C05479=1233.629,-83.711,-36.665,179.745,5.254,148.987
C05480=1233.634,-83.960,-36.654,179.743,5.255,148.988
C05481=1233.639,-84.210,-36.643,179.740,5.254,148.989
C05482=1233.645,-84.460,-36.632,179.738,5.255,148.989
C05483=1233.649,-84.710,-36.620,179.735,5.254,148.990
C05484=1233.655,-84.959,-36.609,179.733,5.254,148.991
C05485=1233.660,-85.209,-36.597,179.730,5.254,148.991
C05486=1233.665,-85.459,-36.587,179.728,5.254,148.992
C05487=1233.670,-85.709,-36.576,179.726,5.254,148.993
C05488=1233.676,-85.958,-36.564,179.724,5.254,148.994
C05489=1233.680,-86.207,-36.553,179.721,5.254,148.994
C05490=1233.685,-86.458,-36.542,179.719,5.254,148.995
C05491=1233.691,-86.707,-36.531,179.716,5.254,148.996
C05492=1233.696,-86.957,-36.519,179.714,5.254,148.996
C05493=1233.701,-87.206,-36.508,179.711,5.254,148.997
C05494=1233.707,-87.457,-36.497,179.709,5.254,148.998
C05495=1233.712,-87.706,-36.486,179.707,5.253,148.999
C05496=1233.716,-87.955,-36.475,179.704,5.254,148.999
C05497=1233.722,-88.206,-36.464,179.702,5.253,149.000
C05498=1233.728,-88.455,-36.453,179.700,5.254,149.001
C05499=1233.732,-88.704,-36.441,179.697,5.253,149.001
C05500=1233.737,-88.954,-36.430,179.695,5.254,149.002
C05501=1233.743,-89.205,-36.419,179.692,5.253,149.003
C05502=1233.748,-89.454,-36.408,179.690,5.253,149.004
C05503=1233.753,-89.704,-36.397,179.688,5.254,149.004
C05504=1233.758,-89.954,-36.386,179.685,5.253,149.005
C05505=1233.764,-90.203,-36.375,179.683,5.254,149.006
C05506=1233.769,-90.453,-36.364,179.681,5.253,149.006
C05507=1233.773,-90.703,-36.353,179.679,5.254,149.007
C05508=1233.779,-90.952,-36.341,179.676,5.253,149.008
C05509=1233.784,-91.202,-36.331,179.674,5.254,149.009
C05510=1233.789,-91.452,-36.319,179.671,5.253,149.009
C05511=1233.795,-91.701,-36.309,179.669,5.253,149.010
C05512=1233.799,-91.951,-36.298,179.666,5.253,149.011
C05513=1233.805,-92.200,-36.286,179.664,5.253,149.011
C05514=1233.810,-92.450,-36.276,179.662,5.253,149.012
C05515=1233.815,-92.700,-36.264,179.659,5.253,149.013
C05516=1233.821,-92.949,-36.254,179.657,5.253,149.014
C05517=1233.826,-93.199,-36.242,179.655,5.253,149.014
C05518=1233.831,-93.450,-36.232,179.652,5.253,149.015
C05519=1233.836,-93.699,-36.221,179.650,5.253,149.016
C05520=1233.841,-93.949,-36.210,179.647,5.253,149.016
C05521=1233.846,-94.198,-36.199,179.645,5.253,149.017
C05522=1233.851,-94.447,-36.188,179.642,5.252,149.018
C05523=1233.857,-94.698,-36.177,179.640,5.253,149.019
C05524=1233.862,-94.947,-36.166,179.638,5.252,149.019
C05525=1233.867,-95.197,-36.155,179.636,5.253,149.020
C05526=1233.872,-95.447,-36.144,179.634,5.253,149.021
C05527=1233.878,-95.696,-36.134,179.631,5.253,149.021
C05528=1233.883,-95.946,-36.123,179.629,5.253,149.022
C05529=1233.889,-96.196,-36.112,179.626,5.253,149.023
C05530=1233.894,-96.446,-36.101,179.624,5.253,149.024
C05531=1233.898,-96.696,-36.090,179.621,5.252,149.024
C05532=1233.904,-96.945,-36.080,179.620,5.252,149.025
C05533=1233.909,-97.195,-36.068,179.617,5.252,149.025
C05534=1233.914,-97.444,-36.058,179.615,5.252,149.026
C05535=1233.919,-97.694,-36.047,179.612,5.252,149.027
C05536=1233.925,-97.943,-36.037,179.610,5.252,149.028
C05537=1233.930,-98.194,-36.026,179.608,5.252,149.028
C05538=1233.936,-98.443,-36.015,179.605,5.252,149.029
C05539=1233.941,-98.693,-36.004,179.603,5.252,149.030
C05540=1233.945,-98.943,-35.993,179.601,5.252,149.030
C05541=1233.951,-99.192,-35.983,179.598,5.252,149.031
C05542=1233.956,-99.443,-35.972,179.596,5.252,149.032
C05543=1233.961,-99.692,-35.961,179.593,5.252,149.033
C05544=1233.966,-99.942,-35.951,179.591,5.252,149.033
C05545=1233.972,-100.213,-35.938,179.588,5.251,149.034
C05546=1233.978,-100.483,-35.928,179.586,5.252,149.035
C05547=1233.983,-100.754,-35.915,179.583,5.252,149.036
C05548=1233.988,-101.025,-35.904,179.581,5.252,149.036
C05549=1233.994,-101.275,-35.894,179.578,5.252,149.037
C05550=1233.999,-101.525,-35.883,179.576,5.252,149.038
C05551=1234.004,-101.774,-35.872,179.574,5.252,149.038
C05552=1234.009,-102.024,-35.861,179.572,5.252,149.039
C05553=1234.015,-102.274,-35.851,179.569,5.251,149.040
C05554=1234.020,-102.524,-35.841,179.567,5.252,149.041
C05555=1234.025,-102.773,-35.830,179.564,5.251,149.041
C05556=1234.030,-103.023,-35.819,179.562,5.252,149.042
C05557=1234.035,-103.272,-35.809,179.559,5.251,149.043
C05558=1234.040,-103.522,-35.798,179.557,5.252,149.043
C05559=1234.046,-103.772,-35.788,179.555,5.252,149.044
C05560=1234.051,-104.022,-35.777,179.552,5.252,149.045
C05561=1234.056,-104.271,-35.767,179.550,5.252,149.046
C05562=1234.061,-104.521,-35.755,179.548,5.251,149.046
C05563=1234.067,-104.771,-35.745,179.546,5.251,149.047
C05564=1234.072,-105.021,-35.735,179.543,5.251,149.048
C05565=1234.077,-105.270,-35.724,179.541,5.251,149.048
C05566=1234.082,-105.520,-35.713,179.539,5.251,149.049
C05567=1234.088,-105.770,-35.703,179.537,5.251,149.050
C05568=1234.093,-106.020,-35.692,179.534,5.251,149.050
C05569=1234.098,-106.269,-35.682,179.532,5.251,149.051
C05570=1234.104,-106.519,-35.672,179.529,5.251,149.052
C05571=1234.108,-106.769,-35.661,179.527,5.251,149.053
C05572=1234.114,-107.018,-35.650,179.525,5.252,149.053
C05573=1234.119,-107.268,-35.640,179.522,5.251,149.054
C05574=1234.125,-107.518,-35.630,179.520,5.251,149.055
C05575=1234.130,-107.768,-35.619,179.517,5.251,149.055
C05576=1234.134,-108.017,-35.609,179.515,5.251,149.056
C05577=1234.139,-108.268,-35.599,179.513,5.251,149.057
C05578=1234.145,-108.516,-35.588,179.511,5.251,149.058
C05579=1234.150,-108.766,-35.578,179.508,5.251,149.058
C05580=1234.155,-109.016,-35.567,179.506,5.251,149.059
C05581=1234.161,-109.266,-35.557,179.504,5.250,149.059
C05582=1234.166,-109.516,-35.546,179.502,5.251,149.060
C05583=1234.172,-109.766,-35.536,179.499,5.250,149.061
C05584=1234.177,-110.016,-35.526,179.497,5.251,149.062
C05585=1234.181,-110.265,-35.516,179.495,5.251,149.062
C05586=1234.187,-110.515,-35.506,179.492,5.251,149.063
C05587=1234.192,-110.764,-35.495,179.490,5.251,149.064
C05588=1234.197,-111.014,-35.484,179.487,5.251,149.064
C05589=1234.202,-111.264,-35.474,179.485,5.251,149.065
C05590=1234.208,-111.514,-35.464,179.482,5.250,149.066
C05591=1234.213,-111.763,-35.453,179.480,5.251,149.067
C05592=1234.218,-112.013,-35.443,179.478,5.250,149.067
C05593=1234.223,-112.263,-35.433,179.476,5.251,149.068
C05594=1234.229,-112.512,-35.423,179.473,5.250,149.069
C05595=1234.234,-112.762,-35.412,179.471,5.251,149.069
C05596=1234.240,-113.012,-35.402,179.469,5.251,149.070
C05597=1234.244,-113.262,-35.392,179.467,5.250,149.071
C05598=1234.249,-113.511,-35.382,179.464,5.251,149.071
C05599=1234.255,-113.761,-35.372,179.462,5.250,149.072
C05600=1234.260,-114.011,-35.361,179.460,5.251,149.073
C05601=1234.266,-114.261,-35.351,179.457,5.250,149.074
C05602=1234.270,-114.510,-35.341,179.455,5.251,149.074
C05603=1234.275,-114.760,-35.331,179.452,5.250,149.075
C05604=1234.281,-115.010,-35.321,179.450,5.250,149.076
C05605=1234.287,-115.259,-35.310,179.448,5.251,149.076
C05606=1234.291,-115.509,-35.300,179.445,5.250,149.077
C05607=1234.296,-115.759,-35.290,179.443,5.251,149.078
C05608=1234.302,-116.008,-35.280,179.441,5.250,149.079
C05609=1234.307,-116.259,-35.269,179.439,5.250,149.079
C05610=1234.312,-116.508,-35.260,179.436,5.250,149.080
C05611=1234.318,-116.758,-35.250,179.434,5.250,149.080
C05612=1234.323,-117.008,-35.240,179.432,5.250,149.081
C05613=1234.328,-117.258,-35.229,179.429,5.250,149.082
C05614=1234.333,-117.507,-35.220,179.427,5.250,149.083
C05615=1234.338,-117.757,-35.209,179.425,5.250,149.083
C05616=1234.344,-118.007,-35.199,179.423,5.250,149.084
C05617=1234.349,-118.256,-35.189,179.420,5.250,149.085
C05618=1234.354,-118.506,-35.179,179.418,5.250,149.085
C05619=1234.360,-118.756,-35.169,179.415,5.250,149.086
C05620=1234.365,-119.006,-35.159,179.413,5.250,149.087
C05621=1234.370,-119.255,-35.150,179.411,5.250,149.087
C05622=1234.375,-119.505,-35.139,179.409,5.250,149.088
C05623=1234.381,-119.755,-35.129,179.406,5.249,149.089
C05624=1234.386,-120.004,-35.119,179.404,5.250,149.090
C05625=1234.391,-120.254,-35.109,179.402,5.250,149.090
C05626=1234.396,-120.505,-35.099,179.399,5.250,149.091
C05627=1234.401,-120.754,-35.090,179.397,5.250,149.092
C05628=1234.407,-121.003,-35.079,179.394,5.250,149.092
C05629=1234.412,-121.254,-35.069,179.392,5.250,149.093
C05630=1234.417,-121.503,-35.059,179.390,5.250,149.094
C05631=1234.423,-121.753,-35.050,179.388,5.250,149.094
C05632=1234.428,-122.002,-35.040,179.385,5.249,149.095
C05633=1234.433,-122.253,-35.029,179.383,5.250,149.096
C05634=1234.438,-122.502,-35.019,179.381,5.250,149.096
C05635=1234.443,-122.752,-35.010,179.378,5.250,149.097
C05636=1234.449,-123.001,-35.000,179.376,5.250,149.098
C05637=1234.454,-123.252,-34.990,179.374,5.250,149.099
C05638=1234.459,-123.501,-34.980,179.372,5.250,149.099
C05639=1234.465,-123.751,-34.970,179.369,5.249,149.100
C05640=1234.470,-124.000,-34.961,179.367,5.249,149.101
C05641=1234.475,-124.251,-34.950,179.365,5.249,149.101
C05642=1234.480,-124.501,-34.941,179.363,5.249,149.102
C05643=1234.485,-124.750,-34.931,179.360,5.250,149.103
C05644=1234.491,-124.999,-34.921,179.358,5.249,149.103
C05645=1234.496,-125.249,-34.911,179.356,5.250,149.104
C05646=1234.501,-125.500,-34.901,179.353,5.249,149.105
C05647=1234.506,-125.749,-34.892,179.351,5.250,149.106
C05648=1234.512,-125.998,-34.882,179.348,5.249,149.106
C05649=1234.091,-126.009,-34.917,179.344,5.252,149.108
C05650=1234.085,-125.759,-34.927,179.347,5.253,149.107
C05651=1234.080,-125.510,-34.937,179.349,5.252,149.107
C05652=1234.074,-125.260,-34.947,179.351,5.253,149.106
C05653=1234.068,-125.010,-34.956,179.353,5.253,149.106
C05654=1234.064,-124.760,-34.966,179.356,5.253,149.105
C05655=1234.058,-124.511,-34.976,179.358,5.253,149.104
C05656=1234.053,-124.261,-34.985,179.360,5.253,149.103
C05657=1234.048,-124.011,-34.996,179.363,5.253,149.103
C05658=1234.043,-123.761,-35.006,179.365,5.253,149.102
C05659=1234.038,-123.512,-35.016,179.368,5.253,149.101
C05660=1234.032,-123.262,-35.025,179.369,5.253,149.101
C05661=1234.027,-123.013,-35.035,179.372,5.253,149.100
C05662=1234.021,-122.763,-35.045,179.374,5.253,149.099
C05663=1234.016,-122.513,-35.056,179.376,5.253,149.099
C05664=1234.011,-122.263,-35.064,179.379,5.253,149.098
C05665=1234.006,-122.013,-35.075,179.381,5.253,149.097
C05666=1234.001,-121.764,-35.084,179.384,5.253,149.096
C05667=1233.996,-121.514,-35.095,179.386,5.253,149.096
C05668=1233.990,-121.264,-35.104,179.388,5.253,149.095
C05669=1233.985,-121.015,-35.114,179.390,5.253,149.094
C05670=1233.980,-120.764,-35.125,179.393,5.254,149.094
C05671=1233.974,-120.515,-35.135,179.395,5.253,149.093
C05672=1233.970,-120.266,-35.144,179.397,5.253,149.092
C05673=1233.964,-120.015,-35.154,179.399,5.253,149.092
C05674=1233.959,-119.765,-35.164,179.402,5.253,149.091
C05675=1233.954,-119.516,-35.174,179.404,5.253,149.090
C05676=1233.948,-119.266,-35.184,179.406,5.253,149.090
C05677=1233.943,-119.017,-35.194,179.409,5.253,149.089
C05678=1233.938,-118.767,-35.204,179.411,5.253,149.088
C05679=1233.932,-118.517,-35.214,179.414,5.254,149.087
C05680=1233.927,-118.267,-35.224,179.415,5.254,149.087
C05681=1233.923,-118.017,-35.234,179.418,5.254,149.086
C05682=1233.917,-117.768,-35.244,179.420,5.254,149.085
C05683=1233.911,-117.518,-35.255,179.422,5.253,149.085
C05684=1233.906,-117.268,-35.265,179.425,5.254,149.084
C05685=1233.902,-117.019,-35.275,179.427,5.253,149.083
C05686=1233.896,-116.769,-35.285,179.430,5.254,149.083
C05687=1233.891,-116.519,-35.296,179.432,5.253,149.082
C05688=1233.886,-116.269,-35.304,179.435,5.254,149.081
C05689=1233.880,-116.019,-35.315,179.437,5.253,149.080
C05690=1233.875,-115.769,-35.325,179.439,5.254,149.080
C05691=1233.870,-115.520,-35.335,179.441,5.254,149.079
C05692=1233.865,-115.270,-35.345,179.443,5.254,149.079
C05693=1233.860,-115.020,-35.356,179.446,5.254,149.078
C05694=1233.854,-114.771,-35.366,179.448,5.254,149.077
C05695=1233.849,-114.521,-35.376,179.450,5.254,149.076
C05696=1233.844,-114.271,-35.387,179.453,5.254,149.076
C05697=1233.839,-114.022,-35.396,179.455,5.254,149.075
C05698=1233.833,-113.772,-35.406,179.457,5.254,149.074
C05699=1233.828,-113.522,-35.417,179.460,5.254,149.073
C05700=1233.822,-113.272,-35.427,179.462,5.254,149.073
C05701=1233.818,-113.023,-35.437,179.465,5.254,149.072
C05702=1233.813,-112.773,-35.447,179.467,5.254,149.071
C05703=1233.807,-112.523,-35.458,179.469,5.253,149.071
C05704=1233.801,-112.274,-35.468,179.471,5.254,149.070
C05705=1233.796,-112.023,-35.478,179.473,5.254,149.069
C05706=1233.791,-111.774,-35.489,179.476,5.254,149.069
C05707=1233.787,-111.524,-35.499,179.478,5.254,149.068
C05708=1233.781,-111.274,-35.509,179.481,5.254,149.067
C05709=1233.775,-111.025,-35.519,179.483,5.254,149.067
C05710=1233.770,-110.775,-35.530,179.485,5.255,149.066
C05711=1233.765,-110.525,-35.540,179.488,5.254,149.065
C05712=1233.760,-110.275,-35.550,179.490,5.255,149.064
C05713=1233.755,-110.026,-35.560,179.492,5.254,149.064
C05714=1233.750,-109.777,-35.571,179.494,5.254,149.063
C05715=1233.745,-109.526,-35.581,179.497,5.254,149.062
C05716=1233.739,-109.277,-35.592,179.499,5.254,149.062
C05717=1233.734,-109.027,-35.602,179.502,5.254,149.061
C05718=1233.728,-108.777,-35.612,179.504,5.254,149.060
C05719=1233.723,-108.528,-35.623,179.506,5.255,149.060
C05720=1233.718,-108.277,-35.633,179.508,5.254,149.059
C05721=1233.712,-108.028,-35.643,179.511,5.255,149.058
C05722=1233.708,-107.779,-35.654,179.513,5.255,149.058
C05723=1233.703,-107.529,-35.664,179.516,5.255,149.057
C05724=1233.698,-107.279,-35.675,179.518,5.255,149.056
C05725=1233.692,-107.029,-35.685,179.520,5.254,149.055
C05726=1233.687,-106.779,-35.696,179.523,5.255,149.055
C05727=1233.681,-106.529,-35.706,179.525,5.254,149.054
C05728=1233.676,-106.280,-35.717,179.527,5.255,149.053
C05729=1233.671,-106.030,-35.727,179.529,5.254,149.053
C05730=1233.666,-105.781,-35.738,179.532,5.255,149.052
C05731=1233.661,-105.530,-35.748,179.534,5.254,149.051
C05732=1233.655,-105.281,-35.758,179.537,5.255,149.050
C05733=1233.650,-105.031,-35.770,179.539,5.255,149.050
C05734=1233.645,-104.782,-35.780,179.542,5.255,149.049
C05735=1233.640,-104.531,-35.790,179.544,5.255,149.048
C05736=1233.634,-104.282,-35.801,179.546,5.255,149.048
C05737=1233.629,-104.032,-35.812,179.548,5.255,149.047
C05738=1233.625,-103.783,-35.822,179.550,5.255,149.046
C05739=1233.620,-103.533,-35.832,179.553,5.255,149.046
C05740=1233.614,-103.283,-35.842,179.555,5.255,149.045
C05741=1233.609,-103.034,-35.854,179.558,5.255,149.044
C05742=1233.604,-102.784,-35.864,179.560,5.255,149.043
C05743=1233.599,-102.534,-35.874,179.562,5.255,149.043
C05744=1233.593,-102.284,-35.885,179.564,5.255,149.042
C05745=1233.588,-102.035,-35.896,179.567,5.255,149.041
C05746=1233.583,-101.785,-35.906,179.569,5.255,149.041
C05747=1233.578,-101.535,-35.917,179.572,5.255,149.040
C05748=1233.572,-101.286,-35.928,179.574,5.255,149.039
C05749=1233.567,-101.035,-35.939,179.577,5.256,149.038
C05750=1233.561,-100.765,-35.950,179.579,5.255,149.038
C05751=1233.555,-100.494,-35.962,179.581,5.256,149.037
C05752=1233.550,-100.223,-35.973,179.584,5.255,149.036
C05753=1233.545,-99.952,-35.985,179.587,5.255,149.035
C05754=1233.539,-99.703,-35.996,179.589,5.255,149.035
C05755=1233.534,-99.452,-36.006,179.591,5.255,149.034
C05756=1233.529,-99.203,-36.017,179.594,5.255,149.033
C05757=1233.524,-98.953,-36.028,179.596,5.256,149.033
C05758=1233.518,-98.704,-36.038,179.598,5.255,149.032
C05759=1233.514,-98.454,-36.049,179.601,5.256,149.031
C05760=1233.508,-98.205,-36.060,179.603,5.255,149.030
C05761=1233.503,-97.954,-36.070,179.606,5.256,149.030
C05762=1233.498,-97.704,-36.082,179.608,5.255,149.029
C05763=1233.492,-97.455,-36.092,179.611,5.256,149.028
C05764=1233.487,-97.205,-36.104,179.613,5.255,149.028
C05765=1233.482,-96.956,-36.114,179.615,5.256,149.027
C05766=1233.477,-96.706,-36.125,179.617,5.256,149.026
C05767=1233.471,-96.456,-36.135,179.620,5.256,149.026
C05768=1233.466,-96.206,-36.146,179.622,5.256,149.025
C05769=1233.462,-95.957,-36.157,179.624,5.256,149.024
C05770=1233.455,-95.707,-36.168,179.626,5.256,149.023
C05771=1233.451,-95.457,-36.179,179.628,5.256,149.023
C05772=1233.445,-95.208,-36.189,179.631,5.256,149.022
C05773=1233.440,-94.958,-36.201,179.633,5.256,149.021
C05774=1233.435,-94.708,-36.211,179.636,5.256,149.021
C05775=1233.430,-94.459,-36.222,179.638,5.256,149.020
C05776=1233.424,-94.208,-36.233,179.641,5.256,149.019
C05777=1233.419,-93.959,-36.244,179.643,5.256,149.019
C05778=1233.414,-93.709,-36.255,179.645,5.256,149.018
C05779=1233.409,-93.459,-36.266,179.648,5.256,149.017
C05780=1233.404,-93.210,-36.276,179.650,5.257,149.016
C05781=1233.399,-92.960,-36.288,179.652,5.256,149.016
C05782=1233.394,-92.710,-36.300,179.655,5.257,149.015
C05783=1233.388,-92.461,-36.310,179.657,5.256,149.014
C05784=1233.383,-92.211,-36.321,179.660,5.257,149.014
C05785=1233.378,-91.962,-36.331,179.662,5.256,149.013
C05786=1233.373,-91.712,-36.343,179.665,5.257,149.012
C05787=1233.367,-91.461,-36.354,179.667,5.257,149.011
C05788=1233.362,-91.213,-36.365,179.669,5.257,149.011
C05789=1233.357,-90.963,-36.376,179.671,5.257,149.010
C05790=1233.352,-90.713,-36.386,179.674,5.257,149.009
C05791=1233.346,-90.463,-36.398,179.676,5.257,149.009
C05792=1233.341,-90.213,-36.409,179.679,5.257,149.008
C05793=1233.337,-89.964,-36.420,179.681,5.257,149.007
C05794=1233.331,-89.715,-36.431,179.684,5.257,149.006
C05795=1233.326,-89.464,-36.442,179.686,5.257,149.006
C05796=1233.321,-89.214,-36.453,179.688,5.257,149.005
C05797=1233.316,-88.966,-36.464,179.690,5.257,149.004
C05798=1233.311,-88.715,-36.475,179.693,5.257,149.004
C05799=1233.305,-88.465,-36.487,179.695,5.257,149.003
C05800=1233.300,-88.216,-36.498,179.697,5.257,149.002
C05801=1233.295,-87.966,-36.508,179.700,5.257,149.001
C05802=1233.290,-87.716,-36.520,179.702,5.257,149.001
C05803=1233.285,-87.467,-36.531,179.705,5.257,149.000
C05804=1233.279,-87.217,-36.542,179.707,5.257,148.999
C05805=1233.275,-86.967,-36.553,179.710,5.257,148.999
C05806=1233.269,-86.717,-36.565,179.712,5.257,148.998
C05807=1233.264,-86.469,-36.576,179.714,5.258,148.997
C05808=1233.259,-86.218,-36.586,179.716,5.257,148.996
C05809=1233.253,-85.968,-36.598,179.719,5.258,148.996
C05810=1233.249,-85.719,-36.609,179.721,5.257,148.995
C05811=1233.243,-85.470,-36.620,179.724,5.258,148.994
C05812=1233.238,-85.219,-36.631,179.726,5.257,148.994
C05813=1233.233,-84.970,-36.643,179.729,5.258,148.993
C05814=1233.228,-84.720,-36.654,179.731,5.258,148.992
C05815=1233.222,-84.471,-36.666,179.733,5.258,148.991
C05816=1233.217,-84.221,-36.676,179.735,5.258,148.991
C05817=1233.212,-83.971,-36.688,179.738,5.258,148.990
C05818=1233.207,-83.721,-36.699,179.740,5.258,148.989
C05819=1233.202,-83.472,-36.710,179.743,5.258,148.989
C05820=1233.196,-83.222,-36.722,179.745,5.258,148.988
C05821=1233.192,-82.973,-36.733,179.748,5.258,148.987
C05822=1233.187,-82.722,-36.744,179.750,5.258,148.986
C05823=1233.181,-82.473,-36.755,179.752,5.258,148.986
C05824=1233.176,-82.223,-36.767,179.754,5.258,148.985
C05825=1233.171,-81.973,-36.779,179.757,5.259,148.984
C05826=1233.166,-81.724,-36.790,179.759,5.258,148.984
C05827=1233.161,-81.474,-36.801,179.762,5.259,148.983
C05828=1233.155,-81.224,-36.812,179.764,5.258,148.982
C05829=1233.150,-80.975,-36.823,179.767,5.259,148.982
C05830=1233.145,-80.725,-36.835,179.769,5.258,148.981
C05831=1233.140,-80.475,-36.847,179.771,5.259,148.980
C05832=1233.134,-80.226,-36.858,179.774,5.259,148.979
C05833=1233.129,-79.976,-36.869,179.776,5.259,148.979
C05834=1233.124,-79.726,-36.881,179.778,5.259,148.978
C05835=1233.119,-79.477,-36.893,179.781,5.259,148.977
C05836=1233.115,-79.227,-36.904,179.783,5.259,148.977
C05837=1233.109,-78.977,-36.916,179.786,5.259,148.976
C05838=1233.104,-78.728,-36.927,179.788,5.259,148.975
C05839=1233.098,-78.478,-36.938,179.791,5.259,148.974
C05840=1233.093,-78.228,-36.949,179.793,5.259,148.974
C05841=1233.088,-77.978,-36.961,179.795,5.259,148.973
C05842=1233.083,-77.729,-36.972,179.797,5.259,148.972
C05843=1233.077,-77.479,-36.984,179.800,5.260,148.972
C05844=1233.073,-77.230,-36.995,179.802,5.259,148.971
C05845=1233.067,-76.980,-37.007,179.805,5.260,148.970
C05846=1233.062,-76.730,-37.018,179.807,5.259,148.969
C05847=1233.057,-76.480,-37.030,179.810,5.260,148.969
C05848=1233.052,-76.231,-37.041,179.812,5.260,148.968
C05849=1233.047,-75.981,-37.053,179.814,5.260,148.967
C05850=1233.041,-75.731,-37.065,179.816,5.260,148.967
C05851=1233.036,-75.482,-37.076,179.819,5.260,148.966
C05852=1233.031,-75.232,-37.088,179.821,5.260,148.965
C05853=1233.026,-74.982,-37.099,179.824,5.260,148.965
C05854=1233.021,-74.712,-37.112,179.826,5.260,148.964
C05855=1233.015,-74.442,-37.125,179.829,5.260,148.963
C05856=1233.010,-74.172,-37.138,179.832,5.260,148.962
C05857=1233.003,-73.902,-37.150,179.834,5.260,148.961
C05858=1232.998,-73.652,-37.162,179.837,5.261,148.961
C05859=1232.993,-73.402,-37.173,179.839,5.260,148.960
C05860=1232.988,-73.152,-37.185,179.841,5.261,148.959
C05861=1232.983,-72.903,-37.197,179.843,5.260,148.959
C05862=1232.978,-72.653,-37.209,179.846,5.261,148.958
C05863=1232.972,-72.403,-37.221,179.848,5.260,148.957
C05864=1232.968,-72.154,-37.232,179.851,5.261,148.956
C05865=1232.962,-71.904,-37.244,179.854,5.261,148.956
C05866=1232.957,-71.654,-37.256,179.856,5.261,148.955
C05867=1232.952,-71.405,-37.267,179.859,5.261,148.954
C05868=1232.946,-71.155,-37.278,179.861,5.261,148.953
C05869=1232.942,-70.906,-37.290,179.864,5.261,148.953
C05870=1232.936,-70.656,-37.302,179.866,5.261,148.952
C05871=1232.931,-70.406,-37.314,179.868,5.261,148.951
C05872=1232.926,-70.156,-37.325,179.870,5.261,148.951
C05873=1232.921,-69.906,-37.337,179.873,5.262,148.950
C05874=1232.916,-69.657,-37.350,179.875,5.261,148.949
C05875=1232.911,-69.407,-37.361,179.878,5.262,148.948
C05876=1232.906,-69.157,-37.373,179.880,5.261,148.948
C05877=1232.900,-68.908,-37.385,179.883,5.262,148.947
C05878=1232.895,-68.658,-37.396,179.885,5.261,148.946
C05879=1232.890,-68.409,-37.409,179.887,5.262,148.946
C05880=1232.885,-68.159,-37.421,179.889,5.262,148.945
C05881=1232.880,-67.909,-37.432,179.892,5.262,148.944
C05882=1232.875,-67.659,-37.444,179.894,5.262,148.944
C05883=1232.870,-67.410,-37.457,179.897,5.262,148.943
C05884=1232.864,-67.161,-37.468,179.899,5.262,148.942
C05885=1232.859,-66.911,-37.479,179.902,5.262,148.941
C05886=1232.854,-66.661,-37.491,179.904,5.262,148.941
C05887=1232.848,-66.412,-37.504,179.906,5.263,148.940
C05888=1232.844,-66.162,-37.515,179.909,5.263,148.939
C05889=1232.838,-65.912,-37.527,179.911,5.263,148.939
C05890=1232.833,-65.663,-37.540,179.914,5.263,148.938
C05891=1232.828,-65.413,-37.552,179.916,5.263,148.937
C05892=1232.823,-65.163,-37.563,179.919,5.263,148.936
C05893=1232.818,-64.914,-37.575,179.921,5.263,148.936
C05894=1232.812,-64.664,-37.587,179.923,5.263,148.935
C05895=1232.807,-64.414,-37.599,179.925,5.263,148.934
C05896=1232.803,-64.165,-37.611,179.928,5.264,148.934
C05897=1232.797,-63.915,-37.623,179.930,5.263,148.933
C05898=1232.792,-63.665,-37.635,179.933,5.263,148.932
C05899=1232.787,-63.416,-37.648,179.935,5.263,148.931
C05900=1232.782,-63.165,-37.660,179.938,5.263,148.931
C05901=1232.777,-62.916,-37.671,179.940,5.263,148.930
C05902=1232.772,-62.666,-37.684,179.943,5.264,148.929
C05903=1232.767,-62.416,-37.696,179.945,5.263,148.928
C05904=1232.762,-62.167,-37.708,179.948,5.264,148.928
C05905=1232.756,-61.917,-37.720,179.950,5.264,148.927
C05906=1232.751,-61.667,-37.731,179.952,5.264,148.926
C05907=1232.746,-61.418,-37.744,179.955,5.264,148.926
C05908=1232.741,-61.168,-37.756,179.957,5.264,148.925
C05909=1232.736,-60.919,-37.768,179.960,5.264,148.924
C05910=1232.730,-60.669,-37.780,179.962,5.264,148.924
C05911=1232.725,-60.420,-37.793,179.964,5.265,148.923
C05912=1232.720,-60.170,-37.804,179.967,5.264,148.922
C05913=1232.715,-59.921,-37.817,179.969,5.265,148.921
C05914=1232.710,-59.671,-37.829,179.971,5.264,148.921
C05915=1232.705,-59.421,-37.841,179.974,5.265,148.920
C05916=1232.699,-59.171,-37.853,179.977,5.265,148.919
C05917=1232.695,-58.921,-37.866,179.979,5.265,148.919
C05918=1232.689,-58.672,-37.878,179.981,5.266,148.918
C05919=1232.685,-58.423,-37.890,179.984,5.265,148.917
C05920=1232.680,-58.173,-37.902,179.986,5.266,148.916
C05921=1232.674,-57.923,-37.915,179.988,5.265,148.916
C05922=1232.669,-57.673,-37.926,179.991,5.266,148.915
C05923=1232.664,-57.424,-37.939,179.993,5.266,148.914
C05924=1232.658,-57.174,-37.951,179.996,5.266,148.913
C05925=1232.653,-56.925,-37.963,179.998,5.265,148.913
C05926=1232.649,-56.674,-37.976,-179.999,5.266,148.912
C05927=1232.643,-56.425,-37.988,-179.996,5.266,148.911
C05928=1232.638,-56.175,-38.001,-179.994,5.266,148.911
C05929=1232.633,-55.926,-38.013,-179.992,5.266,148.910
C05930=1232.628,-55.676,-38.025,-179.990,5.266,148.909
C05931=1232.623,-55.427,-38.037,-179.987,5.267,148.908
C05932=1232.618,-55.177,-38.049,-179.985,5.266,148.908
C05933=1232.613,-54.928,-38.062,-179.982,5.267,148.907
C05934=1232.608,-54.677,-38.074,-179.980,5.266,148.906
C05935=1232.603,-54.428,-38.087,-179.977,5.267,148.906
C05936=1232.597,-54.178,-38.099,-179.975,5.267,148.905
C05937=1232.592,-53.929,-38.111,-179.973,5.267,148.904
C05938=1232.587,-53.679,-38.124,-179.970,5.268,148.904
C05939=1232.582,-53.430,-38.136,-179.968,5.267,148.903
C05940=1232.577,-53.179,-38.149,-179.965,5.268,148.902
C05941=1232.572,-52.930,-38.161,-179.963,5.267,148.901
C05942=1232.567,-52.680,-38.173,-179.960,5.268,148.901
C05943=1232.562,-52.431,-38.186,-179.958,5.268,148.900
C05944=1232.556,-52.182,-38.198,-179.956,5.268,148.899
C05945=1232.551,-51.932,-38.211,-179.953,5.269,148.899
C05946=1232.546,-51.682,-38.223,-179.951,5.268,148.898
C05947=1232.541,-51.432,-38.236,-179.948,5.268,148.897
C05948=1232.536,-51.183,-38.248,-179.946,5.268,148.896
C05949=1232.531,-50.933,-38.260,-179.943,5.268,148.896
C05950=1232.526,-50.684,-38.273,-179.941,5.268,148.895
C05951=1232.521,-50.434,-38.286,-179.938,5.269,148.894
C05952=1232.516,-50.184,-38.299,-179.936,5.268,148.893
C05953=1232.511,-49.934,-38.310,-179.934,5.269,148.893
C05954=1232.505,-49.685,-38.324,-179.931,5.269,148.892
C05955=1232.500,-49.436,-38.336,-179.929,5.269,148.891
C05956=1232.495,-49.186,-38.349,-179.926,5.269,148.891
C05957=1232.490,-48.936,-38.361,-179.924,5.269,148.890
C05958=1232.485,-48.666,-38.375,-179.921,5.270,148.889
C05959=1232.479,-48.397,-38.388,-179.918,5.270,148.888
C05960=1232.473,-48.127,-38.402,-179.916,5.269,148.888
C05961=1232.468,-47.857,-38.416,-179.913,5.270,148.887
C05962=1232.463,-47.607,-38.428,-179.911,5.270,148.886
C05963=1232.458,-47.358,-38.440,-179.909,5.270,148.886
C05964=1232.452,-47.108,-38.454,-179.906,5.271,148.885
C05965=1232.447,-46.858,-38.467,-179.904,5.270,148.884
C05966=1232.442,-46.609,-38.479,-179.901,5.271,148.883
C05967=1232.437,-46.360,-38.492,-179.899,5.270,148.883
C05968=1232.432,-46.110,-38.504,-179.897,5.271,148.882
C05969=1232.427,-45.860,-38.517,-179.893,5.271,148.881
C05970=1232.422,-45.610,-38.529,-179.891,5.271,148.880
C05971=1232.416,-45.361,-38.543,-179.889,5.271,148.880
C05972=1232.411,-45.111,-38.555,-179.887,5.271,148.879
C05973=1232.407,-44.861,-38.568,-179.884,5.271,148.878
C05974=1232.401,-44.612,-38.581,-179.881,5.272,148.878
C05975=1232.396,-44.363,-38.593,-179.879,5.271,148.877
C05976=1232.391,-44.113,-38.606,-179.876,5.272,148.876
C05977=1232.386,-43.863,-38.619,-179.874,5.272,148.875
C05978=1232.381,-43.614,-38.632,-179.872,5.272,148.875
C05979=1232.376,-43.364,-38.645,-179.870,5.272,148.874
C05980=1232.371,-43.114,-38.657,-179.867,5.272,148.873
C05981=1232.366,-42.864,-38.669,-179.864,5.273,148.873
C05982=1232.360,-42.615,-38.683,-179.862,5.273,148.872
C05983=1232.355,-42.365,-38.696,-179.860,5.273,148.871
C05984=1232.350,-42.115,-38.708,-179.857,5.273,148.871
C05985=1232.345,-41.866,-38.721,-179.855,5.273,148.870
C05986=1232.341,-41.616,-38.734,-179.853,5.273,148.869
C05987=1232.335,-41.366,-38.747,-179.850,5.273,148.868
C05988=1232.330,-41.117,-38.760,-179.847,5.274,148.868
C05989=1232.325,-40.867,-38.773,-179.845,5.274,148.867
C05990=1232.320,-40.618,-38.785,-179.842,5.274,148.866
C05991=1232.314,-40.368,-38.798,-179.840,5.273,148.865
C05992=1232.310,-40.119,-38.812,-179.837,5.274,148.865
C05993=1232.305,-39.869,-38.825,-179.835,5.274,148.864
C05994=1232.299,-39.620,-38.838,-179.833,5.274,148.863
C05995=1232.294,-39.370,-38.851,-179.830,5.275,148.863
C05996=1232.289,-39.121,-38.863,-179.828,5.274,148.862
C05997=1232.284,-38.871,-38.876,-179.825,5.275,148.861
C05998=1232.279,-38.621,-38.890,-179.823,5.275,148.861
C05999=1232.274,-38.372,-38.902,-179.820,5.275,148.860
C06000=1232.269,-38.122,-38.915,-179.818,5.275,148.859
C06001=1232.263,-37.872,-38.928,-179.816,5.275,148.858
C06002=1232.258,-37.623,-38.941,-179.813,5.276,148.858
C06003=1232.254,-37.373,-38.954,-179.810,5.276,148.857
C06004=1232.248,-37.124,-38.968,-179.808,5.276,148.856
C06005=1232.243,-36.874,-38.980,-179.806,5.276,148.856
C06006=1232.238,-36.624,-38.993,-179.804,5.276,148.855
C06007=1232.233,-36.375,-39.007,-179.801,5.276,148.854
C06008=1232.227,-36.125,-39.019,-179.798,5.277,148.854
C06009=1232.223,-35.875,-39.032,-179.796,5.277,148.853
C06010=1232.217,-35.626,-39.045,-179.793,5.277,148.852
C06011=1232.213,-35.376,-39.059,-179.791,5.276,148.851
C06012=1232.208,-35.127,-39.072,-179.788,5.277,148.850
C06013=1232.202,-34.877,-39.085,-179.786,5.277,148.850
C06014=1232.197,-34.627,-39.098,-179.784,5.277,148.849
C06015=1232.191,-34.378,-39.111,-179.781,5.278,148.848
C06016=1232.187,-34.128,-39.125,-179.779,5.277,148.848
C06017=1232.182,-33.879,-39.137,-179.776,5.278,148.847
C06018=1232.177,-33.629,-39.151,-179.773,5.278,148.846
C06019=1232.172,-33.379,-39.163,-179.771,5.278,148.846
C06020=1232.166,-33.130,-39.177,-179.769,5.278,148.845
C06021=1232.162,-32.880,-39.190,-179.767,5.278,148.844
C06022=1232.157,-32.631,-39.203,-179.764,5.279,148.843
C06023=1232.151,-32.381,-39.216,-179.761,5.279,148.843
C06024=1232.146,-32.132,-39.230,-179.759,5.279,148.842
C06025=1232.141,-31.882,-39.243,-179.757,5.279,148.841
C06026=1232.136,-31.632,-39.256,-179.754,5.279,148.841
C06027=1232.131,-31.383,-39.270,-179.752,5.280,148.840
C06028=1232.126,-31.133,-39.283,-179.749,5.280,148.839
C06029=1232.121,-30.883,-39.296,-179.747,5.280,148.839
C06030=1232.116,-30.634,-39.309,-179.744,5.280,148.838
C06031=1232.111,-30.384,-39.323,-179.741,5.280,148.837
C06032=1232.106,-30.135,-39.336,-179.739,5.280,148.836
C06033=1232.100,-29.885,-39.348,-179.736,5.281,148.836
C06034=1232.095,-29.636,-39.363,-179.734,5.280,148.835
C06035=1232.090,-29.386,-39.375,-179.732,5.281,148.834
C06036=1232.085,-29.136,-39.390,-179.729,5.281,148.833
C06037=1232.080,-28.887,-39.402,-179.727,5.281,148.833
C06038=1232.075,-28.637,-39.416,-179.724,5.281,148.832
C06039=1232.070,-28.388,-39.429,-179.722,5.281,148.831
C06040=1232.065,-28.138,-39.443,-179.720,5.282,148.831
C06041=1232.060,-27.888,-39.455,-179.717,5.282,148.830
C06042=1232.055,-27.639,-39.470,-179.715,5.282,148.829
C06043=1232.050,-27.389,-39.483,-179.712,5.282,148.829
C06044=1232.045,-27.140,-39.496,-179.710,5.283,148.828
C06045=1232.040,-26.889,-39.510,-179.707,5.283,148.827
C06046=1232.035,-26.641,-39.523,-179.705,5.283,148.827
C06047=1232.029,-26.390,-39.537,-179.703,5.283,148.826
C06048=1232.025,-26.142,-39.550,-179.700,5.283,148.825
C06049=1232.019,-25.891,-39.564,-179.697,5.284,148.824
C06050=1232.014,-25.642,-39.576,-179.695,5.283,148.824
C06051=1232.009,-25.392,-39.591,-179.693,5.284,148.823
C06052=1232.004,-25.143,-39.603,-179.690,5.285,148.822
C06053=1231.999,-24.893,-39.617,-179.687,5.284,148.821
C06054=1231.993,-24.644,-39.631,-179.685,5.284,148.821
C06055=1231.989,-24.394,-39.644,-179.682,5.285,148.820
C06056=1231.984,-24.144,-39.658,-179.680,5.285,148.819
C06057=1231.979,-23.895,-39.671,-179.677,5.285,148.819
C06058=1231.974,-23.645,-39.685,-179.675,5.285,148.818
C06059=1231.968,-23.396,-39.699,-179.673,5.285,148.817
C06060=1231.964,-23.147,-39.712,-179.670,5.286,148.817
C06061=1231.959,-22.896,-39.726,-179.668,5.285,148.816
C06062=1231.953,-22.627,-39.741,-179.665,5.286,148.815
C06063=1231.948,-22.358,-39.755,-179.663,5.286,148.814
C06064=1231.943,-22.089,-39.770,-179.659,5.287,148.814
C06065=1231.937,-21.820,-39.785,-179.657,5.286,148.813
C06066=1231.931,-21.570,-39.798,-179.655,5.287,148.812
C06067=1231.927,-21.321,-39.812,-179.652,5.287,148.811
C06068=1231.921,-21.071,-39.825,-179.650,5.287,148.811
C06069=1231.916,-20.821,-39.839,-179.647,5.288,148.810
C06070=1231.912,-20.572,-39.853,-179.645,5.288,148.809
C06071=1231.906,-20.322,-39.866,-179.642,5.288,148.809
C06072=1231.901,-20.072,-39.880,-179.640,5.288,148.808
C06073=1231.896,-19.823,-39.893,-179.637,5.289,148.807
C06074=1231.891,-19.573,-39.907,-179.635,5.288,148.807
C06075=1231.886,-19.324,-39.922,-179.632,5.289,148.806
C06076=1231.880,-19.074,-39.935,-179.630,5.290,148.805
C06077=1231.876,-18.825,-39.949,-179.627,5.289,148.804
C06078=1231.871,-18.575,-39.963,-179.625,5.289,148.804
C06079=1231.865,-18.325,-39.976,-179.622,5.289,148.803
C06080=1231.861,-18.076,-39.990,-179.620,5.290,148.802
C06081=1231.856,-17.827,-40.004,-179.617,5.290,148.801
C06082=1231.851,-17.577,-40.018,-179.615,5.290,148.801
C06083=1231.845,-17.327,-40.031,-179.612,5.290,148.800
C06084=1231.841,-17.078,-40.045,-179.610,5.291,148.799
C06085=1231.836,-16.828,-40.059,-179.608,5.291,148.799
C06086=1231.831,-16.579,-40.073,-179.605,5.291,148.798
C06087=1231.825,-16.329,-40.086,-179.602,5.292,148.797
C06088=1231.820,-16.079,-40.101,-179.600,5.291,148.797
C06089=1231.816,-15.830,-40.114,-179.598,5.292,148.796
C06090=1231.811,-15.580,-40.129,-179.595,5.292,148.795
C06091=1231.805,-15.331,-40.142,-179.593,5.292,148.795
C06092=1231.800,-15.081,-40.156,-179.590,5.292,148.794
C06093=1231.795,-14.831,-40.170,-179.588,5.293,148.793
C06094=1231.790,-14.583,-40.184,-179.585,5.293,148.792
C06095=1231.785,-14.333,-40.198,-179.583,5.293,148.792
C06096=1231.780,-14.083,-40.212,-179.580,5.294,148.791
C06097=1231.774,-13.834,-40.226,-179.578,5.293,148.790
C06098=1231.769,-13.584,-40.240,-179.575,5.294,148.790
C06099=1231.765,-13.334,-40.254,-179.573,5.294,148.789
C06100=1231.760,-13.085,-40.268,-179.571,5.294,148.788
C06101=1231.755,-12.836,-40.282,-179.568,5.295,148.788
C06102=1231.749,-12.585,-40.295,-179.565,5.295,148.787
C06103=1231.744,-12.336,-40.310,-179.563,5.295,148.786
C06104=1231.739,-12.087,-40.323,-179.560,5.295,148.785
C06105=1231.734,-11.837,-40.338,-179.557,5.296,148.785
C06106=1231.730,-11.588,-40.351,-179.555,5.295,148.784
C06107=1231.725,-11.338,-40.366,-179.553,5.296,148.783
C06108=1231.719,-11.089,-40.380,-179.550,5.296,148.782
C06109=1231.714,-10.839,-40.394,-179.548,5.296,148.782
C06110=1231.709,-10.589,-40.408,-179.545,5.297,148.781
C06111=1231.704,-10.339,-40.422,-179.543,5.297,148.780
C06112=1231.698,-10.090,-40.436,-179.541,5.297,148.780
C06113=1231.693,-9.840,-40.450,-179.538,5.297,148.779
C06114=1231.688,-9.591,-40.464,-179.535,5.298,148.778
C06115=1231.684,-9.341,-40.478,-179.533,5.298,148.778
C06116=1231.679,-9.092,-40.492,-179.531,5.298,148.777
C06117=1231.674,-8.843,-40.506,-179.528,5.299,148.776
C06118=1231.669,-8.593,-40.520,-179.525,5.299,148.776
C06119=1231.664,-8.343,-40.535,-179.523,5.299,148.775
C06120=1231.659,-8.093,-40.549,-179.521,5.299,148.774
C06121=1231.653,-7.844,-40.563,-179.518,5.300,148.773
C06122=1231.648,-7.595,-40.577,-179.516,5.300,148.773
C06123=1231.643,-7.345,-40.591,-179.513,5.300,148.772
C06124=1231.638,-7.095,-40.606,-179.510,5.301,148.771
C06125=1231.634,-6.846,-40.620,-179.508,5.300,148.771
C06126=1231.629,-6.596,-40.634,-179.506,5.301,148.770
C06127=1231.623,-6.347,-40.648,-179.503,5.301,148.769
C06128=1231.618,-6.097,-40.662,-179.501,5.301,148.769
C06129=1231.613,-5.848,-40.677,-179.498,5.302,148.768
C06130=1231.608,-5.598,-40.692,-179.496,5.302,148.767
C06131=1231.603,-5.349,-40.706,-179.494,5.302,148.767
C06132=1231.598,-5.100,-40.720,-179.491,5.302,148.766
C06133=1231.593,-4.850,-40.734,-179.488,5.303,148.765
C06134=1231.588,-4.600,-40.748,-179.486,5.303,148.765
C06135=1231.583,-4.350,-40.763,-179.484,5.303,148.764
C06136=1231.578,-4.101,-40.777,-179.480,5.303,148.763
C06137=1231.573,-3.851,-40.791,-179.478,5.304,148.762
C06138=1231.568,-3.601,-40.805,-179.476,5.304,148.762
C06139=1231.563,-3.353,-40.820,-179.473,5.304,148.761
C06140=1231.558,-3.103,-40.834,-179.470,5.305,148.760
C06141=1231.553,-2.853,-40.849,-179.468,5.304,148.759
C06142=1231.548,-2.604,-40.863,-179.466,5.305,148.759
C06143=1231.543,-2.354,-40.877,-179.463,5.305,148.758
C06144=1231.538,-2.104,-40.891,-179.460,5.306,148.757
C06145=1231.534,-1.855,-40.906,-179.458,5.306,148.757
C06146=1231.529,-1.606,-40.921,-179.456,5.306,148.756
C06147=1231.522,-1.356,-40.935,-179.453,5.307,148.755
C06148=1231.517,-1.107,-40.950,-179.451,5.306,148.755
C06149=1231.512,-0.857,-40.964,-179.448,5.307,148.754
C06150=1231.508,-0.608,-40.979,-179.446,5.307,148.753
C06151=1231.503,-0.358,-40.993,-179.443,5.308,148.753
C06152=1231.498,-0.108,-41.007,-179.441,5.308,148.752
C06153=1231.493,0.141,-41.022,-179.438,5.308,148.751
C06154=1231.488,0.391,-41.037,-179.436,5.309,148.750
C06155=1231.483,0.641,-41.052,-179.433,5.308,148.750
C06156=1231.478,0.890,-41.066,-179.431,5.309,148.749
C06157=1231.472,1.139,-41.080,-179.428,5.309,148.748
C06158=1231.467,1.388,-41.095,-179.426,5.309,148.748
C06159=1231.462,1.638,-41.109,-179.423,5.310,148.747
C06160=1231.457,1.888,-41.123,-179.421,5.310,148.746
C06161=1231.453,2.137,-41.138,-179.418,5.311,148.746
C06162=1231.447,2.387,-41.153,-179.416,5.310,148.745
C06163=1231.442,2.637,-41.167,-179.413,5.311,148.744
C06164=1231.437,2.886,-41.182,-179.411,5.312,148.744
C06165=1231.433,3.135,-41.197,-179.408,5.312,148.743
C06166=1231.427,3.404,-41.212,-179.406,5.312,148.742
C06167=1231.422,3.673,-41.229,-179.403,5.312,148.741
C06168=1231.416,3.942,-41.244,-179.400,5.313,148.741
C06169=1231.411,4.211,-41.260,-179.398,5.313,148.740
C06170=1231.406,4.461,-41.275,-179.395,5.314,148.739
C06171=1231.401,4.711,-41.289,-179.393,5.313,148.739
C06172=1231.396,4.960,-41.304,-179.390,5.314,148.738
C06173=1231.391,5.209,-41.319,-179.388,5.314,148.737
C06174=1231.386,5.458,-41.333,-179.385,5.315,148.736
C06175=1231.381,5.709,-41.348,-179.383,5.315,148.736
C06176=1231.375,5.958,-41.362,-179.380,5.315,148.735
C06177=1231.370,6.207,-41.377,-179.378,5.316,148.734
C06178=1231.366,6.456,-41.392,-179.375,5.316,148.734
C06179=1231.360,6.706,-41.407,-179.373,5.316,148.733
C06180=1231.355,6.955,-41.421,-179.370,5.316,148.732
C06181=1231.351,7.205,-41.437,-179.367,5.317,148.732
C06182=1231.345,7.455,-41.452,-179.365,5.318,148.731
C06183=1231.341,7.704,-41.467,-179.363,5.317,148.730
C06184=1231.336,7.954,-41.481,-179.360,5.318,148.730
C06185=1231.331,8.203,-41.496,-179.357,5.318,148.729
C06186=1231.326,8.453,-41.511,-179.355,5.318,148.728
C06187=1231.321,8.702,-41.526,-179.353,5.319,148.728
C06188=1231.316,8.952,-41.540,-179.350,5.319,148.727
C06189=1231.311,9.201,-41.556,-179.347,5.320,148.726
C06190=1231.306,9.451,-41.570,-179.345,5.319,148.725
C06191=1231.301,9.700,-41.585,-179.343,5.320,148.725
C06192=1231.295,9.950,-41.600,-179.340,5.320,148.724
C06193=1231.291,10.199,-41.615,-179.337,5.321,148.723
C06194=1231.286,10.448,-41.630,-179.335,5.321,148.723
C06195=1231.280,10.698,-41.645,-179.333,5.321,148.722
C06196=1231.276,10.947,-41.660,-179.330,5.322,148.721
C06197=1231.271,11.197,-41.674,-179.327,5.322,148.721
C06198=1231.265,11.447,-41.689,-179.325,5.322,148.720
C06199=1231.261,11.696,-41.704,-179.323,5.323,148.719
C06200=1231.255,11.946,-41.719,-179.320,5.323,148.719
C06201=1231.250,12.195,-41.734,-179.317,5.324,148.718
C06202=1231.246,12.445,-41.749,-179.315,5.323,148.717
C06203=1231.241,12.695,-41.765,-179.313,5.324,148.717
C06204=1231.236,12.944,-41.780,-179.310,5.324,148.716
C06205=1231.230,13.194,-41.794,-179.307,5.325,148.715
C06206=1231.226,13.443,-41.809,-179.305,5.325,148.715
C06207=1231.221,13.692,-41.824,-179.303,5.325,148.714
C06208=1231.215,13.942,-41.839,-179.300,5.326,148.713
C06209=1231.211,14.191,-41.854,-179.297,5.326,148.712
C06210=1231.205,14.440,-41.870,-179.295,5.327,148.712
C06211=1231.200,14.690,-41.884,-179.293,5.327,148.711
C06212=1231.195,14.940,-41.900,-179.290,5.327,148.710
C06213=1231.191,15.189,-41.915,-179.287,5.328,148.710
C06214=1231.185,15.439,-41.931,-179.285,5.328,148.709
C06215=1231.180,15.688,-41.945,-179.283,5.328,148.708
C06216=1231.176,15.938,-41.960,-179.280,5.329,148.708
C06217=1231.170,16.187,-41.976,-179.277,5.329,148.707
C06218=1231.166,16.436,-41.991,-179.275,5.330,148.706
C06219=1231.160,16.686,-42.005,-179.273,5.329,148.706
C06220=1231.156,16.936,-42.021,-179.270,5.330,148.705
C06221=1231.151,17.185,-42.036,-179.267,5.330,148.704
C06222=1231.146,17.434,-42.051,-179.265,5.331,148.704
C06223=1231.140,17.684,-42.066,-179.262,5.331,148.703
C06224=1231.136,17.933,-42.081,-179.260,5.331,148.702
C06225=1231.130,18.183,-42.097,-179.257,5.332,148.702
C06226=1231.126,18.433,-42.112,-179.255,5.332,148.701
C06227=1231.121,18.682,-42.128,-179.252,5.333,148.700
C06228=1231.115,18.931,-42.143,-179.250,5.333,148.699
C06229=1231.110,19.181,-42.158,-179.247,5.333,148.699
C06230=1231.105,19.431,-42.173,-179.245,5.334,148.698
C06231=1231.101,19.680,-42.189,-179.242,5.334,148.697
C06232=1231.096,19.930,-42.204,-179.239,5.335,148.697
C06233=1231.091,20.179,-42.219,-179.237,5.334,148.696
C06234=1231.086,20.428,-42.235,-179.235,5.335,148.695
C06235=1231.081,20.677,-42.250,-179.232,5.336,148.695
C06236=1231.076,20.927,-42.265,-179.229,5.336,148.694
C06237=1231.071,21.177,-42.281,-179.227,5.337,148.693
C06238=1231.066,21.427,-42.296,-179.225,5.336,148.693
C06239=1231.060,21.676,-42.311,-179.222,5.337,148.692
C06240=1231.056,21.925,-42.326,-179.219,5.338,148.691
C06241=1231.051,22.175,-42.342,-179.217,5.338,148.691
C06242=1231.046,22.425,-42.358,-179.215,5.338,148.690
C06243=1231.041,22.674,-42.373,-179.212,5.338,148.689
C06244=1231.036,22.923,-42.388,-179.209,5.339,148.689
C06245=1231.031,23.173,-42.404,-179.207,5.339,148.688
C06246=1231.026,23.422,-42.419,-179.204,5.340,148.687
C06247=1231.021,23.672,-42.435,-179.202,5.340,148.687
C06248=1231.016,23.921,-42.450,-179.200,5.341,148.686
C06249=1231.011,24.171,-42.466,-179.197,5.341,148.685
C06250=1231.006,24.420,-42.481,-179.194,5.342,148.685
C06251=1231.001,24.669,-42.496,-179.192,5.342,148.684
C06252=1230.996,24.919,-42.512,-179.190,5.342,148.683
C06253=1230.991,25.169,-42.528,-179.187,5.343,148.683
C06254=1230.986,25.418,-42.543,-179.184,5.343,148.682
C06255=1230.981,25.667,-42.558,-179.182,5.344,148.681
C06256=1230.976,25.917,-42.574,-179.179,5.344,148.681
C06257=1230.971,26.167,-42.590,-179.176,5.345,148.680
C06258=1230.966,26.416,-42.605,-179.174,5.344,148.679
C06259=1230.961,26.665,-42.621,-179.172,5.345,148.679
C06260=1230.956,26.915,-42.637,-179.169,5.346,148.678
C06261=1230.952,27.164,-42.652,-179.166,5.346,148.677
C06262=1230.946,27.413,-42.668,-179.164,5.347,148.677
C06263=1230.941,27.663,-42.683,-179.162,5.346,148.676
C06264=1230.936,27.913,-42.699,-179.159,5.347,148.675
C06265=1230.932,28.162,-42.714,-179.156,5.348,148.675
C06266=1230.926,28.411,-42.730,-179.154,5.348,148.674
C06267=1230.921,28.661,-42.746,-179.151,5.349,148.673
C06268=1230.916,28.910,-42.762,-179.149,5.348,148.672
C06269=1230.912,29.159,-42.777,-179.146,5.349,148.672
C06270=1230.907,29.428,-42.795,-179.144,5.349,148.671
C06271=1230.901,29.697,-42.812,-179.141,5.350,148.670
C06272=1230.896,29.965,-42.829,-179.139,5.351,148.670
C06273=1230.890,30.235,-42.845,-179.136,5.351,148.669
C06274=1230.885,30.483,-42.861,-179.133,5.352,148.668
C06275=1230.881,30.733,-42.877,-179.131,5.352,148.668
C06276=1230.875,30.983,-42.892,-179.128,5.353,148.667
C06277=1230.870,31.232,-42.908,-179.126,5.353,148.666
C06278=1230.865,31.481,-42.924,-179.123,5.353,148.666
C06279=1230.860,31.731,-42.940,-179.121,5.354,148.665
C06280=1230.856,31.981,-42.955,-179.118,5.354,148.664
C06281=1230.850,32.230,-42.971,-179.115,5.355,148.664
C06282=1230.845,32.479,-42.987,-179.113,5.355,148.663
C06283=1230.841,32.729,-43.003,-179.111,5.355,148.662
C06284=1230.835,32.978,-43.019,-179.108,5.356,148.662
C06285=1230.830,33.228,-43.034,-179.105,5.356,148.661
C06286=1230.825,33.477,-43.051,-179.103,5.357,148.660
C06287=1230.821,33.726,-43.066,-179.100,5.357,148.660
C06288=1230.816,33.976,-43.082,-179.097,5.358,148.659
C06289=1230.811,34.225,-43.098,-179.095,5.358,148.658
C06290=1230.805,34.475,-43.114,-179.093,5.358,148.658
C06291=1230.801,34.725,-43.130,-179.090,5.359,148.657
C06292=1230.796,34.973,-43.146,-179.088,5.360,148.656
C06293=1230.791,35.224,-43.162,-179.085,5.360,148.656
C06294=1230.785,35.473,-43.178,-179.083,5.361,148.655
C06295=1230.781,35.722,-43.194,-179.080,5.361,148.654
C06296=1230.776,35.972,-43.210,-179.078,5.361,148.654
C06297=1230.771,36.220,-43.226,-179.075,5.362,148.653
C06298=1230.766,36.470,-43.242,-179.073,5.362,148.652
C06299=1230.761,36.720,-43.257,-179.070,5.363,148.652
C06300=1230.757,36.969,-43.274,-179.067,5.363,148.651
C06301=1230.751,37.219,-43.289,-179.065,5.364,148.650
C06302=1230.747,37.468,-43.306,-179.062,5.364,148.650
C06303=1230.741,37.718,-43.322,-179.060,5.364,148.649
C06304=1230.737,37.967,-43.338,-179.057,5.365,148.648
C06305=1230.731,38.216,-43.354,-179.055,5.365,148.648
C06306=1230.726,38.465,-43.370,-179.052,5.366,148.647
C06307=1230.722,38.715,-43.386,-179.049,5.366,148.646
C06308=1230.716,38.965,-43.402,-179.047,5.367,148.646
C06309=1230.712,39.214,-43.418,-179.045,5.368,148.645
C06310=1230.706,39.464,-43.434,-179.043,5.368,148.645
C06311=1230.702,39.713,-43.451,-179.040,5.368,148.644
C06312=1230.696,39.963,-43.466,-179.037,5.369,148.643
C06313=1230.692,40.212,-43.483,-179.035,5.369,148.642
C06314=1230.687,40.461,-43.499,-179.032,5.370,148.642
C06315=1230.682,40.711,-43.515,-179.029,5.370,148.641
C06316=1230.677,40.960,-43.532,-179.027,5.371,148.640
C06317=1230.672,41.210,-43.548,-179.024,5.372,148.640
C06318=1230.667,41.459,-43.564,-179.022,5.371,148.639
C06319=1230.662,41.709,-43.580,-179.019,5.372,148.638
C06320=1230.657,41.957,-43.596,-179.017,5.372,148.638
C06321=1230.652,42.208,-43.613,-179.015,5.373,148.637
C06322=1230.647,42.457,-43.629,-179.012,5.374,148.637
C06323=1230.642,42.706,-43.646,-179.009,5.374,148.636
C06324=1230.637,42.956,-43.661,-179.007,5.375,148.635
C06325=1230.632,43.205,-43.678,-179.004,5.376,148.635
C06326=1230.627,43.454,-43.694,-179.002,5.375,148.634
C06327=1230.622,43.704,-43.710,-178.999,5.376,148.633
C06328=1230.618,43.953,-43.727,-178.997,5.376,148.633
C06329=1230.613,44.203,-43.742,-178.994,5.377,148.632
C06330=1230.608,44.452,-43.759,-178.991,5.378,148.631
C06331=1230.602,44.701,-43.776,-178.989,5.378,148.631
C06332=1230.598,44.951,-43.792,-178.986,5.379,148.630
C06333=1230.592,45.200,-43.808,-178.984,5.380,148.629
C06334=1230.588,45.450,-43.825,-178.981,5.380,148.629
C06335=1230.583,45.699,-43.841,-178.979,5.380,148.628
C06336=1230.578,45.949,-43.857,-178.977,5.381,148.627
C06337=1230.574,46.198,-43.874,-178.974,5.381,148.627
C06338=1230.568,46.447,-43.891,-178.971,5.382,148.626
C06339=1230.563,46.697,-43.907,-178.969,5.382,148.625
C06340=1230.558,46.946,-43.923,-178.966,5.383,148.625
C06341=1230.553,47.196,-43.940,-178.963,5.383,148.624
C06342=1230.549,47.445,-43.956,-178.961,5.384,148.623
C06343=1230.544,47.694,-43.972,-178.958,5.385,148.623
C06344=1230.538,47.944,-43.989,-178.957,5.385,148.622
C06345=1230.533,48.193,-44.005,-178.954,5.385,148.622
C06346=1230.529,48.443,-44.022,-178.951,5.386,148.621
C06347=1230.524,48.692,-44.039,-178.949,5.386,148.620
C06348=1230.519,48.941,-44.054,-178.946,5.387,148.620
C06349=1230.514,49.191,-44.072,-178.943,5.388,148.619
C06350=1230.509,49.441,-44.088,-178.941,5.388,148.618
C06351=1230.504,49.689,-44.105,-178.938,5.389,148.618
C06352=1230.500,49.939,-44.121,-178.935,5.389,148.617
C06353=1230.494,50.188,-44.138,-178.933,5.390,148.617
C06354=1230.489,50.438,-44.154,-178.931,5.391,148.616
C06355=1230.485,50.688,-44.171,-178.929,5.390,148.615
C06356=1230.480,50.936,-44.187,-178.926,5.391,148.614
C06357=1230.474,51.186,-44.204,-178.923,5.392,148.614
C06358=1230.470,51.436,-44.221,-178.921,5.392,148.613
C06359=1230.465,51.684,-44.237,-178.918,5.393,148.612
C06360=1230.460,51.934,-44.255,-178.915,5.393,148.612
C06361=1230.455,52.184,-44.271,-178.913,5.394,148.611
C06362=1230.450,52.433,-44.288,-178.911,5.395,148.611
C06363=1230.445,52.682,-44.304,-178.908,5.395,148.610
C06364=1230.440,52.932,-44.321,-178.905,5.396,148.609
C06365=1230.435,53.181,-44.337,-178.903,5.397,148.609
C06366=1230.430,53.431,-44.354,-178.900,5.397,148.608
C06367=1230.425,53.681,-44.371,-178.898,5.397,148.607
C06368=1230.421,53.930,-44.388,-178.895,5.397,148.607
C06369=1230.416,54.179,-44.404,-178.893,5.398,148.606
C06370=1230.410,54.429,-44.421,-178.890,5.399,148.605
C06371=1230.406,54.678,-44.438,-178.888,5.400,148.605
C06372=1230.401,54.927,-44.454,-178.885,5.400,148.604
C06373=1230.396,55.177,-44.471,-178.883,5.401,148.604
C06374=1230.391,55.445,-44.490,-178.880,5.401,148.603
C06375=1230.385,55.713,-44.508,-178.877,5.402,148.602
C06376=1230.380,55.982,-44.526,-178.875,5.402,148.602
C06377=1230.374,56.250,-44.544,-178.872,5.403,148.601
C06378=1230.370,56.500,-44.561,-178.870,5.404,148.600
C06379=1230.365,56.749,-44.578,-178.867,5.404,148.600
C06380=1230.360,56.998,-44.595,-178.864,5.405,148.599
C06381=1230.355,57.248,-44.611,-178.862,5.405,148.598
C06382=1230.350,57.497,-44.629,-178.859,5.406,148.598
C06383=1230.345,57.747,-44.645,-178.856,5.406,148.597
C06384=1230.341,57.995,-44.662,-178.854,5.407,148.596
C06385=1230.335,58.245,-44.679,-178.851,5.408,148.596
C06386=1230.331,58.494,-44.696,-178.849,5.409,148.595
C06387=1230.326,58.744,-44.713,-178.846,5.409,148.594
C06388=1230.321,58.993,-44.730,-178.844,5.410,148.594
C06389=1230.315,59.243,-44.747,-178.841,5.410,148.593
C06390=1230.311,59.492,-44.764,-178.838,5.411,148.592
C06391=1230.306,59.741,-44.782,-178.836,5.411,148.592
C06392=1230.302,59.991,-44.798,-178.833,5.412,148.591
C06393=1230.296,60.240,-44.815,-178.831,5.413,148.591
C06394=1230.291,60.489,-44.832,-178.828,5.414,148.590
C06395=1230.286,60.739,-44.849,-178.826,5.413,148.589
C06396=1230.282,60.988,-44.866,-178.824,5.414,148.589
C06397=1230.276,61.237,-44.883,-178.821,5.414,148.588
C06398=1230.272,61.487,-44.900,-178.818,5.415,148.587
C06399=1230.266,61.736,-44.917,-178.816,5.416,148.587
C06400=1230.262,61.986,-44.934,-178.814,5.417,148.586
C06401=1230.257,62.235,-44.952,-178.811,5.417,148.586
C06402=1230.252,62.485,-44.969,-178.808,5.418,148.585
C06403=1230.247,62.734,-44.986,-178.806,5.418,148.584
C06404=1230.242,62.983,-45.003,-178.803,5.419,148.584
C06405=1230.237,63.232,-45.020,-178.801,5.419,148.583
C06406=1230.233,63.482,-45.037,-178.798,5.420,148.582
C06407=1230.228,63.732,-45.054,-178.796,5.421,148.582
C06408=1230.223,63.981,-45.072,-178.793,5.422,148.581
C06409=1230.218,64.230,-45.088,-178.790,5.422,148.581
C06410=1230.212,64.479,-45.106,-178.788,5.423,148.580
C06411=1230.208,64.728,-45.123,-178.785,5.423,148.579
C06412=1230.203,64.978,-45.140,-178.783,5.424,148.579
C06413=1230.198,65.228,-45.158,-178.780,5.425,148.578
C06414=1230.194,65.477,-45.175,-178.778,5.425,148.577
C06415=1230.188,65.727,-45.192,-178.775,5.426,148.577
C06416=1230.184,65.975,-45.210,-178.773,5.427,148.576
C06417=1230.178,66.224,-45.227,-178.770,5.427,148.575
C06418=1230.173,66.474,-45.244,-178.767,5.428,148.575
C06419=1230.169,66.723,-45.261,-178.765,5.429,148.574
C06420=1230.164,66.973,-45.278,-178.763,5.429,148.574
C06421=1230.159,67.222,-45.296,-178.760,5.430,148.573
C06422=1230.154,67.472,-45.313,-178.757,5.430,148.572
C06423=1230.149,67.721,-45.330,-178.755,5.431,148.572
C06424=1230.144,67.971,-45.348,-178.752,5.432,148.571
C06425=1230.140,68.220,-45.365,-178.750,5.433,148.571
C06426=1230.135,68.469,-45.383,-178.747,5.433,148.570
C06427=1230.129,68.718,-45.400,-178.745,5.434,148.569
C06428=1230.125,68.967,-45.417,-178.742,5.434,148.569
C06429=1230.120,69.217,-45.435,-178.739,5.435,148.568
C06430=1230.115,69.466,-45.453,-178.737,5.435,148.567
C06431=1230.110,69.716,-45.469,-178.735,5.436,148.567
C06432=1230.105,69.965,-45.487,-178.732,5.437,148.566
C06433=1230.100,70.215,-45.504,-178.729,5.438,148.566
C06434=1230.096,70.463,-45.522,-178.727,5.438,148.565
C06435=1230.091,70.713,-45.539,-178.724,5.439,148.564
C06436=1230.086,70.962,-45.557,-178.722,5.440,148.564
C06437=1230.081,71.212,-45.575,-178.719,5.440,148.563
C06438=1230.076,71.461,-45.592,-178.717,5.441,148.562
C06439=1230.071,71.710,-45.610,-178.714,5.441,148.562
C06440=1230.066,71.960,-45.627,-178.711,5.442,148.561
C06441=1230.061,72.209,-45.645,-178.709,5.443,148.560
C06442=1230.057,72.459,-45.662,-178.707,5.444,148.560
C06443=1230.052,72.708,-45.680,-178.704,5.444,148.559
C06444=1230.047,72.957,-45.698,-178.701,5.445,148.559
C06445=1230.042,73.207,-45.715,-178.699,5.445,148.558
C06446=1230.037,73.456,-45.733,-178.696,5.446,148.557
C06447=1230.033,73.705,-45.750,-178.694,5.447,148.557
C06448=1230.027,73.955,-45.767,-178.691,5.448,148.556
C06449=1230.023,74.204,-45.785,-178.689,5.448,148.556
C06450=1230.018,74.453,-45.803,-178.686,5.449,148.555
C06451=1230.012,74.703,-45.821,-178.684,5.449,148.554
C06452=1230.008,74.952,-45.839,-178.681,5.450,148.554
C06453=1230.003,75.201,-45.856,-178.679,5.451,148.553
C06454=1229.998,75.451,-45.873,-178.676,5.451,148.553
C06455=1229.993,75.700,-45.891,-178.673,5.452,148.552
C06456=1229.988,75.949,-45.909,-178.671,5.453,148.551
C06457=1229.983,76.199,-45.927,-178.669,5.454,148.551
C06458=1229.978,76.448,-45.944,-178.666,5.454,148.550
C06459=1229.973,76.697,-45.962,-178.663,5.455,148.550
C06460=1229.969,76.946,-45.980,-178.661,5.455,148.549
C06461=1229.964,77.195,-45.998,-178.658,5.456,148.548
C06462=1229.959,77.445,-46.015,-178.656,5.457,148.548
C06463=1229.954,77.694,-46.033,-178.653,5.457,148.547
C06464=1229.949,77.943,-46.051,-178.651,5.458,148.546
C06465=1229.944,78.193,-46.069,-178.648,5.459,148.546
C06466=1229.939,78.442,-46.086,-178.645,5.460,148.545
C06467=1229.934,78.692,-46.104,-178.643,5.461,148.545
C06468=1229.930,78.941,-46.123,-178.640,5.462,148.544
C06469=1229.925,79.191,-46.141,-178.638,5.462,148.543
C06470=1229.920,79.440,-46.159,-178.635,5.463,148.543
C06471=1229.916,79.689,-46.176,-178.633,5.464,148.542
C06472=1229.911,79.938,-46.193,-178.630,5.464,148.542
C06473=1229.906,80.188,-46.211,-178.628,5.465,148.541
C06474=1229.901,80.437,-46.229,-178.625,5.466,148.540
C06475=1229.896,80.686,-46.247,-178.622,5.466,148.540
C06476=1229.891,80.935,-46.265,-178.620,5.467,148.539
C06477=1229.886,81.184,-46.283,-178.618,5.468,148.539
C06478=1229.881,81.453,-46.303,-178.615,5.468,148.538
C06479=1229.875,81.721,-46.323,-178.612,5.470,148.537
C06480=1229.870,81.990,-46.341,-178.609,5.470,148.537
C06481=1229.865,82.258,-46.361,-178.607,5.471,148.536
C06482=1229.860,82.507,-46.379,-178.604,5.471,148.535
C06483=1229.855,82.757,-46.397,-178.601,5.472,148.535
C06484=1229.851,83.006,-46.415,-178.599,5.473,148.534
C06485=1229.846,83.256,-46.433,-178.597,5.474,148.534
C06486=1229.841,83.505,-46.451,-178.594,5.474,148.533
C06487=1229.836,83.754,-46.469,-178.591,5.475,148.532
C06488=1229.831,84.003,-46.487,-178.589,5.476,148.532
C06489=1229.826,84.252,-46.505,-178.586,5.477,148.531
C06490=1229.822,84.502,-46.523,-178.583,5.478,148.531
C06491=1229.817,84.751,-46.541,-178.581,5.478,148.530
C06492=1229.812,85.001,-46.559,-178.579,5.479,148.530
C06493=1229.807,85.250,-46.577,-178.576,5.480,148.529
C06494=1229.802,85.499,-46.595,-178.573,5.481,148.528
C06495=1229.797,85.748,-46.613,-178.571,5.481,148.528
C06496=1229.792,85.998,-46.632,-178.569,5.482,148.527
C06497=1229.787,86.247,-46.650,-178.566,5.483,148.526
C06498=1229.783,86.496,-46.669,-178.563,5.483,148.526
C06499=1229.778,86.745,-46.687,-178.561,5.484,148.525
C06500=1229.773,86.994,-46.705,-178.559,5.485,148.525
C06501=1229.768,87.244,-46.723,-178.555,5.486,148.524
C06502=1229.763,87.493,-46.741,-178.553,5.487,148.523
C06503=1229.759,87.743,-46.759,-178.550,5.488,148.523
C06504=1229.753,87.992,-46.778,-178.548,5.488,148.522
C06505=1229.749,88.242,-46.796,-178.545,5.489,148.522
C06506=1229.744,88.491,-46.815,-178.543,5.490,148.521
C06507=1229.739,88.740,-46.833,-178.540,5.490,148.520
C06508=1229.734,88.989,-46.851,-178.538,5.491,148.520
C06509=1229.729,89.238,-46.869,-178.535,5.492,148.519
C06510=1229.724,89.488,-46.887,-178.533,5.492,148.519
C06511=1229.719,89.737,-46.905,-178.530,5.493,148.518
C06512=1229.715,89.986,-46.924,-178.527,5.495,148.518
C06513=1229.710,90.235,-46.942,-178.525,5.495,148.517
C06514=1229.705,90.485,-46.960,-178.522,5.496,148.516
C06515=1229.700,90.735,-46.979,-178.520,5.497,148.516
C06516=1229.695,90.983,-46.998,-178.517,5.498,148.515
C06517=1229.690,91.232,-47.016,-178.515,5.498,148.515
C06518=1229.686,91.482,-47.034,-178.512,5.499,148.514
C06519=1229.680,91.732,-47.053,-178.510,5.499,148.513
C06520=1229.676,91.980,-47.071,-178.508,5.500,148.513
C06521=1229.671,92.230,-47.090,-178.504,5.502,148.512
C06522=1229.667,92.479,-47.108,-178.502,5.502,148.512
C06523=1229.661,92.728,-47.127,-178.500,5.503,148.511
C06524=1229.656,92.977,-47.145,-178.497,5.504,148.510
C06525=1229.652,93.227,-47.163,-178.494,5.505,148.510
C06526=1229.647,93.476,-47.182,-178.492,5.505,148.509
C06527=1229.642,93.725,-47.201,-178.490,5.506,148.509
C06528=1229.637,93.975,-47.219,-178.487,5.507,148.508
C06529=1229.633,94.224,-47.238,-178.484,5.508,148.507
C06530=1229.627,94.473,-47.256,-178.482,5.509,148.507
C06531=1229.623,94.723,-47.275,-178.479,5.510,148.506
C06532=1229.618,94.972,-47.293,-178.476,5.510,148.506
C06533=1229.613,95.221,-47.311,-178.474,5.511,148.505
C06534=1229.609,95.470,-47.331,-178.472,5.512,148.505
C06535=1229.604,95.719,-47.349,-178.469,5.513,148.504
C06536=1229.599,95.969,-47.367,-178.466,5.513,148.503
C06537=1229.594,96.218,-47.386,-178.464,5.515,148.503
C06538=1229.589,96.467,-47.404,-178.461,5.516,148.502
C06539=1229.584,96.716,-47.424,-178.458,5.516,148.502
C06540=1229.579,96.966,-47.442,-178.456,5.517,148.501
C06541=1229.575,97.215,-47.461,-178.454,5.518,148.501
C06542=1229.569,97.464,-47.479,-178.451,5.518,148.500
C06543=1229.565,97.713,-47.498,-178.449,5.519,148.499
C06544=1229.560,97.963,-47.516,-178.446,5.521,148.499
C06545=1229.555,98.212,-47.536,-178.443,5.521,148.498
C06546=1229.551,98.461,-47.554,-178.441,5.522,148.498
C06547=1229.545,98.710,-47.573,-178.438,5.523,148.497
C06548=1229.541,98.960,-47.592,-178.436,5.523,148.497
C06549=1229.536,99.209,-47.611,-178.433,5.524,148.496
C06550=1229.531,99.458,-47.629,-178.431,5.525,148.495
C06551=1229.527,99.707,-47.648,-178.428,5.526,148.495
C06552=1229.521,99.957,-47.667,-178.425,5.527,148.494
C06553=1229.517,100.206,-47.686,-178.423,5.528,148.494
C06554=1229.512,100.455,-47.705,-178.421,5.529,148.493
C06555=1229.507,100.705,-47.723,-178.418,5.529,148.492
C06556=1229.502,100.954,-47.743,-178.415,5.530,148.492
C06557=1229.497,101.203,-47.761,-178.413,5.532,148.491
C06558=1229.492,101.452,-47.780,-178.410,5.532,148.491
C06559=1229.488,101.701,-47.799,-178.407,5.533,148.490
C06560=1229.483,101.951,-47.818,-178.405,5.534,148.490
C06561=1229.478,102.200,-47.837,-178.403,5.534,148.489
C06562=1229.473,102.449,-47.856,-178.400,5.535,148.488
C06563=1229.468,102.699,-47.874,-178.397,5.537,148.488
C06564=1229.463,102.947,-47.893,-178.395,5.538,148.487
C06565=1229.459,103.197,-47.913,-178.392,5.538,148.487
C06566=1229.453,103.446,-47.931,-178.390,5.539,148.486
C06567=1229.449,103.695,-47.950,-178.387,5.540,148.486
C06568=1229.444,103.944,-47.969,-178.385,5.540,148.485
C06569=1229.440,104.194,-47.988,-178.382,5.542,148.485
C06570=1229.434,104.443,-48.007,-178.379,5.543,148.484
C06571=1229.430,104.692,-48.026,-178.377,5.543,148.483
C06572=1229.425,104.941,-48.045,-178.375,5.544,148.483
C06573=1229.421,105.191,-48.064,-178.372,5.545,148.482
C06574=1229.415,105.440,-48.083,-178.370,5.546,148.482
C06575=1229.411,105.689,-48.103,-178.367,5.547,148.481
C06576=1229.406,105.938,-48.121,-178.364,5.548,148.481
C06577=1229.401,106.188,-48.140,-178.362,5.549,148.480
C06578=1229.396,106.437,-48.159,-178.359,5.550,148.480
C06579=1229.392,106.686,-48.179,-178.357,5.550,148.479
C06580=1229.386,106.935,-48.198,-178.354,5.552,148.478
C06581=1229.382,107.184,-48.217,-178.352,5.553,148.478
C06582=1229.377,107.453,-48.237,-178.349,5.553,148.477
C06583=1229.372,107.722,-48.258,-178.346,5.555,148.477
C06584=1229.366,107.990,-48.279,-178.343,5.555,148.476
C06585=1229.361,108.258,-48.300,-178.341,5.556,148.475
C06586=1229.356,108.507,-48.318,-178.338,5.557,148.475
C06587=1229.352,108.757,-48.338,-178.335,5.558,148.474
C06588=1229.347,109.007,-48.357,-178.333,5.559,148.474
C06589=1229.342,109.255,-48.376,-178.330,5.560,148.473
C06590=1229.337,109.505,-48.396,-178.328,5.560,148.473
C06591=1229.332,109.754,-48.415,-178.325,5.561,148.472
C06592=1229.328,110.003,-48.434,-178.323,5.563,148.471
C06593=1229.323,110.252,-48.453,-178.320,5.563,148.471
C06594=1229.318,110.501,-48.473,-178.317,5.564,148.470
C06595=1229.313,110.751,-48.493,-178.315,5.565,148.470
C06596=1229.309,110.999,-48.511,-178.312,5.567,148.469
C06597=1229.304,111.249,-48.531,-178.310,5.567,148.469
C06598=1229.299,111.498,-48.550,-178.307,5.568,148.468
C06599=1229.295,111.747,-48.569,-178.305,5.569,148.467
C06600=1229.289,111.996,-48.589,-178.303,5.570,148.467
C06601=1229.284,112.246,-48.608,-178.299,5.571,148.466
C06602=1229.280,112.495,-48.628,-178.297,5.572,148.466
C06603=1229.275,112.744,-48.647,-178.295,5.573,148.465
C06604=1229.270,112.993,-48.666,-178.292,5.573,148.465
C06605=1229.265,113.242,-48.686,-178.289,5.575,148.464
C06606=1229.260,113.492,-48.705,-178.287,5.576,148.464
C06607=1229.256,113.741,-48.725,-178.284,5.576,148.463
C06608=1229.251,113.990,-48.744,-178.282,5.577,148.463
C06609=1229.246,114.239,-48.763,-178.279,5.578,148.462
C06610=1229.241,114.489,-48.783,-178.276,5.579,148.461
C06611=1229.236,114.738,-48.802,-178.274,5.580,148.461
C06612=1229.231,114.987,-48.822,-178.272,5.581,148.460
C06613=1229.227,115.237,-48.841,-178.269,5.582,148.460
C06614=1229.222,115.485,-48.861,-178.266,5.583,148.459
C06615=1229.218,115.734,-48.881,-178.264,5.584,148.459
C06616=1229.212,115.983,-48.900,-178.262,5.585,148.458
C06617=1229.207,116.233,-48.919,-178.259,5.586,148.458
C06618=1229.203,116.482,-48.939,-178.256,5.587,148.457
C06619=1229.198,116.731,-48.958,-178.254,5.588,148.457
C06620=1229.194,116.980,-48.978,-178.251,5.589,148.456
C06621=1229.189,117.229,-48.998,-178.249,5.590,148.455
C06622=1229.184,117.479,-49.017,-178.246,5.591,148.455
C06623=1229.179,117.728,-49.037,-178.244,5.592,148.454
C06624=1229.174,117.977,-49.056,-178.241,5.593,148.454
C06625=1229.170,118.226,-49.077,-178.238,5.593,148.453
C06626=1229.164,118.475,-49.096,-178.236,5.595,148.453
C06627=1229.160,118.725,-49.116,-178.233,5.596,148.452
C06628=1229.155,118.974,-49.135,-178.231,5.597,148.452
C06629=1229.151,119.222,-49.155,-178.228,5.597,148.451
C06630=1229.146,119.472,-49.174,-178.225,5.599,148.450
C06631=1229.141,119.722,-49.194,-178.223,5.600,148.450
C06632=1229.136,119.971,-49.214,-178.220,5.600,148.449
C06633=1229.131,120.219,-49.234,-178.218,5.601,148.449
C06634=1229.127,120.469,-49.253,-178.215,5.603,148.448
C06635=1229.122,120.718,-49.273,-178.213,5.604,148.448
C06636=1229.117,120.967,-49.293,-178.210,5.604,148.447
C06637=1229.112,121.216,-49.313,-178.207,5.606,148.447
C06638=1229.107,121.466,-49.332,-178.205,5.607,148.446
C06639=1229.103,121.715,-49.353,-178.203,5.608,148.446
C06640=1229.098,121.964,-49.372,-178.200,5.608,148.445
C06641=1229.093,122.213,-49.392,-178.197,5.610,148.445
C06642=1229.088,122.462,-49.412,-178.195,5.611,148.444
C06643=1229.084,122.712,-49.432,-178.193,5.612,148.444
C06644=1229.079,122.961,-49.452,-178.190,5.612,148.443
C06645=1229.074,123.210,-49.471,-178.187,5.614,148.443
C06646=1229.069,123.459,-49.491,-178.185,5.615,148.442
C06647=1229.065,123.708,-49.511,-178.182,5.615,148.441
C06648=1229.060,123.958,-49.531,-178.179,5.617,148.441
C06649=1229.055,124.206,-49.551,-178.177,5.618,148.440
C06650=1229.050,124.455,-49.571,-178.175,5.619,148.440
C06651=1229.046,124.704,-49.591,-178.172,5.619,148.439
C06652=1229.041,124.954,-49.611,-178.169,5.621,148.439
C06653=1229.036,125.203,-49.631,-178.167,5.622,148.438
C06654=1229.030,125.452,-49.651,-178.165,5.623,148.438
C06655=1229.026,125.701,-49.671,-178.161,5.624,148.437
C06656=1229.021,125.951,-49.691,-178.159,5.625,148.437
C06657=1229.017,126.200,-49.711,-178.157,5.626,148.436
C06658=1229.012,126.449,-49.731,-178.154,5.627,148.436
C06659=1229.008,126.698,-49.751,-178.151,5.628,148.435
C06660=1229.002,126.947,-49.771,-178.149,5.629,148.434
C06661=1228.998,127.196,-49.791,-178.147,5.630,148.434
C06662=1228.993,127.445,-49.812,-178.144,5.631,148.433
C06663=1228.988,127.695,-49.832,-178.141,5.632,148.433
C06664=1228.983,127.944,-49.852,-178.139,5.633,148.432
C06665=1228.979,128.193,-49.872,-178.136,5.634,148.432
C06666=1228.974,128.442,-49.892,-178.134,5.635,148.431
C06667=1228.969,128.690,-49.912,-178.131,5.636,148.431
C06668=1228.965,128.940,-49.932,-178.128,5.638,148.430
C06669=1228.960,129.189,-49.952,-178.126,5.638,148.430
C06670=1228.955,129.439,-49.972,-178.124,5.639,148.429
C06671=1228.950,129.688,-49.993,-178.120,5.641,148.429
C06672=1228.946,129.937,-50.013,-178.118,5.642,148.428
C06673=1228.941,130.186,-50.033,-178.116,5.643,148.428
C06674=1228.937,130.435,-50.053,-178.113,5.644,148.427
C06675=1228.931,130.685,-50.074,-178.110,5.645,148.427
C06676=1228.926,130.933,-50.093,-178.108,5.646,148.426
C06677=1228.922,131.182,-50.114,-178.105,5.647,148.426
C06678=1228.917,131.431,-50.134,-178.103,5.648,148.425
C06679=1228.912,131.681,-50.155,-178.100,5.649,148.425
C06680=1228.907,131.930,-50.175,-178.097,5.650,148.424
C06681=1228.903,132.179,-50.195,-178.095,5.651,148.424
C06682=1228.898,132.428,-50.216,-178.093,5.652,148.423
C06683=1228.893,132.677,-50.237,-178.090,5.654,148.423
C06684=1228.888,132.927,-50.256,-178.087,5.655,148.422
C06685=1228.884,133.176,-50.277,-178.085,5.656,148.422
C06686=1228.879,133.444,-50.299,-178.082,5.657,148.421
C06687=1228.873,133.713,-50.321,-178.079,5.658,148.420
C06688=1228.868,133.981,-50.342,-178.077,5.659,148.420
C06689=1228.863,134.251,-50.365,-178.074,5.660,148.419
C06690=1228.859,134.500,-50.385,-178.071,5.662,148.419
C06691=1228.854,134.749,-50.406,-178.069,5.663,148.418
C06692=1228.849,134.998,-50.426,-178.066,5.663,148.418
C06693=1228.844,135.246,-50.446,-178.064,5.665,148.417
C06694=1228.839,135.495,-50.467,-178.061,5.666,148.417
C06695=1228.835,135.744,-50.488,-178.059,5.667,148.416
C06696=1228.830,135.994,-50.507,-178.056,5.668,148.416
C06697=1228.825,136.243,-50.528,-178.054,5.669,148.415
C06698=1228.820,136.492,-50.549,-178.051,5.670,148.415
C06699=1228.816,136.741,-50.569,-178.048,5.672,148.414
C06700=1228.811,136.990,-50.590,-178.046,5.672,148.414
C06701=1228.806,137.239,-50.610,-178.043,5.674,148.413
C06702=1228.801,137.489,-50.631,-178.040,5.675,148.413
C06703=1228.797,137.738,-50.652,-178.038,5.676,148.412
C06704=1228.792,137.986,-50.672,-178.035,5.677,148.412
C06705=1228.787,138.236,-50.693,-178.033,5.678,148.411
C06706=1228.783,138.485,-50.713,-178.031,5.679,148.411
C06707=1228.777,138.734,-50.734,-178.028,5.680,148.410
C06708=1228.774,138.984,-50.755,-178.026,5.681,148.410
C06709=1228.769,139.233,-50.775,-178.023,5.683,148.409
C06710=1228.764,139.482,-50.796,-178.020,5.684,148.409
C06711=1228.760,139.731,-50.817,-178.018,5.685,148.408
C06712=1228.754,139.980,-50.838,-178.015,5.686,148.408
C06713=1228.750,140.229,-50.858,-178.013,5.687,148.407
C06714=1228.745,140.478,-50.879,-178.010,5.688,148.407
C06715=1228.740,140.727,-50.899,-178.007,5.689,148.406
C06716=1228.735,140.976,-50.920,-178.005,5.690,148.406
C06717=1228.731,141.225,-50.941,-178.002,5.692,148.405
C06718=1228.726,141.474,-50.962,-178.000,5.693,148.405
C06719=1228.721,141.723,-50.983,-177.997,5.694,148.404
C06720=1228.716,141.972,-51.004,-177.995,5.695,148.404
C06721=1228.712,142.221,-51.024,-177.992,5.696,148.403
C06722=1228.707,142.470,-51.045,-177.989,5.698,148.403
C06723=1228.703,142.720,-51.066,-177.987,5.699,148.402
C06724=1228.698,142.969,-51.087,-177.985,5.699,148.402
C06725=1228.693,143.218,-51.107,-177.982,5.701,148.401
C06726=1228.688,143.467,-51.129,-177.979,5.702,148.401
C06727=1228.684,143.716,-51.149,-177.977,5.704,148.400
C06728=1228.679,143.965,-51.170,-177.974,5.704,148.400
C06729=1228.674,144.214,-51.191,-177.972,5.705,148.399
C06730=1228.669,144.463,-51.212,-177.969,5.707,148.399
C06731=1228.664,144.712,-51.233,-177.967,5.708,148.398
C06732=1228.660,144.962,-51.254,-177.964,5.709,148.398
C06733=1228.655,145.211,-51.275,-177.962,5.710,148.397
C06734=1228.651,145.460,-51.295,-177.959,5.711,148.397
C06735=1228.646,145.709,-51.317,-177.956,5.713,148.396
C06736=1228.641,145.958,-51.338,-177.954,5.714,148.396
C06737=1228.636,146.207,-51.358,-177.951,5.715,148.395
C06738=1228.631,146.455,-51.380,-177.949,5.716,148.395
C06739=1228.628,146.705,-51.401,-177.946,5.717,148.394
C06740=1228.622,146.954,-51.422,-177.944,5.719,148.394
C06741=1228.617,147.204,-51.443,-177.941,5.719,148.393
C06742=1228.613,147.452,-51.464,-177.938,5.721,148.393
C06743=1228.608,147.701,-51.485,-177.936,5.722,148.392
C06744=1228.603,147.950,-51.506,-177.933,5.724,148.392
C06745=1228.599,148.199,-51.527,-177.931,5.725,148.391
C06746=1228.594,148.449,-51.548,-177.928,5.725,148.391
C06747=1228.589,148.697,-51.570,-177.926,5.727,148.390
C06748=1228.585,148.946,-51.590,-177.923,5.728,148.390
C06749=1228.580,149.196,-51.611,-177.920,5.730,148.389
C06750=1228.575,149.445,-51.633,-177.918,5.730,148.389
C06751=1228.570,149.694,-51.654,-177.915,5.732,148.388
C06752=1228.566,149.942,-51.675,-177.913,5.733,148.388
C06753=1228.561,150.192,-51.696,-177.910,5.735,148.387
C06754=1228.557,150.441,-51.718,-177.908,5.736,148.387
C06755=1228.552,150.690,-51.739,-177.905,5.736,148.386
C06756=1228.547,150.939,-51.760,-177.903,5.738,148.386
C06757=1228.542,151.188,-51.781,-177.900,5.739,148.385
C06758=1228.537,151.437,-51.802,-177.897,5.740,148.385
C06759=1228.533,151.686,-51.824,-177.895,5.741,148.385
C06760=1228.528,151.935,-51.845,-177.892,5.743,148.384
C06761=1228.523,152.184,-51.866,-177.890,5.744,148.384
C06762=1228.518,152.433,-51.887,-177.887,5.745,148.383
C06763=1228.514,152.683,-51.909,-177.885,5.746,148.383
C06764=1228.509,152.932,-51.930,-177.883,5.747,148.382
C06765=1228.505,153.180,-51.951,-177.879,5.749,148.382
C06766=1228.500,153.429,-51.973,-177.877,5.750,148.381
C06767=1228.495,153.679,-51.994,-177.874,5.751,148.381
C06768=1228.490,153.928,-52.016,-177.872,5.752,148.380
C06769=1228.486,154.176,-52.037,-177.869,5.754,148.380
C06770=1228.482,154.426,-52.059,-177.867,5.755,148.379
C06771=1228.477,154.674,-52.080,-177.864,5.757,148.379
C06772=1228.471,154.924,-52.101,-177.862,5.757,148.378
C06773=1228.467,155.172,-52.123,-177.859,5.759,148.378
C06774=1228.462,155.422,-52.144,-177.857,5.760,148.378
C06775=1228.457,155.671,-52.166,-177.854,5.762,148.377
C06776=1228.453,155.919,-52.187,-177.852,5.763,148.377
C06777=1228.448,156.169,-52.208,-177.848,5.764,148.376
C06778=1228.444,156.418,-52.230,-177.846,5.765,148.376
C06779=1228.439,156.667,-52.252,-177.844,5.767,148.375
C06780=1228.434,156.916,-52.273,-177.841,5.768,148.375
C06781=1228.429,157.165,-52.295,-177.839,5.769,148.374
C06782=1228.424,157.414,-52.316,-177.836,5.770,148.374
C06783=1228.420,157.663,-52.338,-177.834,5.771,148.373
C06784=1228.415,157.912,-52.359,-177.831,5.773,148.373
C06785=1228.410,158.161,-52.381,-177.828,5.774,148.372
C06786=1228.406,158.410,-52.403,-177.826,5.775,148.372
C06787=1228.401,158.659,-52.425,-177.824,5.776,148.371
C06788=1228.396,158.908,-52.446,-177.821,5.778,148.371
C06789=1228.392,159.157,-52.467,-177.818,5.779,148.370
C06790=1228.387,159.426,-52.491,-177.815,5.780,148.370
C06791=1228.382,159.695,-52.515,-177.813,5.782,148.369
C06792=1228.377,159.964,-52.537,-177.809,5.784,148.369
C06793=1228.372,160.233,-52.562,-177.807,5.785,148.368
C06794=1228.367,160.483,-52.583,-177.804,5.786,148.368
C06795=1228.362,160.732,-52.605,-177.802,5.787,148.368
C06796=1228.357,160.980,-52.626,-177.799,5.789,148.367
C06797=1228.353,161.230,-52.648,-177.797,5.790,148.367
C06798=1228.348,161.478,-52.670,-177.794,5.791,148.366
C06799=1228.344,161.728,-52.692,-177.792,5.792,148.366
C06800=1228.339,161.976,-52.714,-177.789,5.794,148.365
C06801=1228.334,162.225,-52.735,-177.787,5.795,148.365
C06802=1228.330,162.475,-52.757,-177.784,5.797,148.364
C06803=1228.325,162.724,-52.778,-177.782,5.797,148.364
C06804=1228.320,162.973,-52.800,-177.779,5.799,148.363
C06805=1228.316,163.222,-52.822,-177.776,5.800,148.363
C06806=1228.311,163.471,-52.844,-177.774,5.802,148.362
C06807=1228.306,163.720,-52.866,-177.772,5.803,148.362
C06808=1228.301,163.969,-52.888,-177.769,5.804,148.361
C06809=1228.297,164.218,-52.910,-177.766,5.805,148.361
C06810=1228.292,164.467,-52.932,-177.764,5.807,148.361
C06811=1228.287,164.716,-52.954,-177.761,5.809,148.360
C06812=1228.283,164.964,-52.976,-177.759,5.810,148.360
C06813=1228.278,165.214,-52.998,-177.756,5.811,148.359
C06814=1228.273,165.462,-53.019,-177.753,5.812,148.359
C06815=1228.269,165.712,-53.041,-177.751,5.814,148.358
C06816=1228.264,165.961,-53.064,-177.749,5.815,148.358
C06817=1228.259,166.210,-53.086,-177.745,5.816,148.357
C06818=1228.255,166.458,-53.108,-177.743,5.817,148.357
C06819=1228.250,166.707,-53.130,-177.741,5.819,148.357
C06820=1228.246,166.956,-53.152,-177.738,5.820,148.356
C06821=1228.241,167.205,-53.174,-177.735,5.822,148.356
C06822=1228.236,167.454,-53.196,-177.733,5.823,148.355
C06823=1228.231,167.704,-53.218,-177.730,5.824,148.355
C06824=1228.227,167.952,-53.240,-177.727,5.826,148.354
C06825=1228.222,168.202,-53.262,-177.725,5.827,148.354
C06826=1228.217,168.450,-53.284,-177.723,5.829,148.354
C06827=1228.213,168.699,-53.307,-177.720,5.830,148.353
C06828=1228.208,168.948,-53.329,-177.717,5.831,148.353
C06829=1228.204,169.197,-53.351,-177.715,5.832,148.352
C06830=1228.199,169.446,-53.372,-177.712,5.834,148.352
C06831=1228.194,169.695,-53.394,-177.710,5.835,148.351
C06832=1228.189,169.944,-53.417,-177.707,5.837,148.351
C06833=1228.185,170.193,-53.439,-177.704,5.838,148.350
C06834=1228.181,170.442,-53.461,-177.702,5.839,148.350
C06835=1228.175,170.691,-53.484,-177.700,5.841,148.350
C06836=1228.171,170.940,-53.507,-177.697,5.842,148.349
C06837=1228.166,171.189,-53.528,-177.694,5.844,148.349
C06838=1228.162,171.438,-53.550,-177.692,5.845,148.348
C06839=1228.156,171.687,-53.573,-177.690,5.846,148.348
C06840=1228.152,171.936,-53.595,-177.686,5.848,148.347
C06841=1228.148,172.185,-53.617,-177.684,5.849,148.347
C06842=1228.143,172.434,-53.640,-177.682,5.851,148.347
C06843=1228.139,172.683,-53.662,-177.679,5.851,148.346
C06844=1228.134,172.931,-53.684,-177.676,5.853,148.346
C06845=1228.129,173.181,-53.707,-177.674,5.854,148.345
C06846=1228.125,173.430,-53.729,-177.672,5.856,148.345
C06847=1228.120,173.678,-53.751,-177.669,5.858,148.344
C06848=1228.115,173.928,-53.774,-177.667,5.859,148.344
C06849=1228.110,174.176,-53.796,-177.664,5.860,148.343
C06850=1228.106,174.425,-53.818,-177.661,5.861,148.343
C06851=1228.101,174.674,-53.842,-177.659,5.863,148.343
C06852=1228.096,174.923,-53.863,-177.656,5.865,148.342
C06853=1228.091,175.173,-53.886,-177.654,5.866,148.342
C06854=1228.087,175.421,-53.909,-177.651,5.867,148.341
C06855=1228.083,175.670,-53.930,-177.649,5.868,148.341
C06856=1228.078,175.919,-53.954,-177.646,5.870,148.340
C06857=1228.073,176.168,-53.975,-177.643,5.872,148.340
C06858=1228.068,176.417,-53.999,-177.641,5.873,148.339
C06859=1228.064,176.666,-54.021,-177.638,5.874,148.339
C06860=1228.059,176.914,-54.044,-177.636,5.875,148.339
C06861=1228.054,177.164,-54.066,-177.633,5.877,148.338
C06862=1228.051,177.412,-54.089,-177.630,5.879,148.338
C06863=1228.046,177.662,-54.111,-177.628,5.880,148.337
C06864=1228.041,177.910,-54.134,-177.626,5.882,148.337
C06865=1228.036,178.160,-54.156,-177.623,5.882,148.336
C06866=1228.032,178.409,-54.179,-177.620,5.884,148.336
C06867=1228.026,178.657,-54.201,-177.618,5.886,148.336
C06868=1228.022,178.906,-54.224,-177.616,5.887,148.335
C06869=1228.017,179.156,-54.247,-177.612,5.888,148.335
C06870=1228.013,179.404,-54.269,-177.610,5.890,148.334
C06871=1228.008,179.653,-54.293,-177.608,5.891,148.334
C06872=1228.004,179.902,-54.315,-177.605,5.893,148.334
C06873=1227.999,180.151,-54.338,-177.602,5.894,148.333
C06874=1227.995,180.399,-54.360,-177.600,5.896,148.333
C06875=1227.990,180.649,-54.383,-177.597,5.898,148.332
C06876=1227.986,180.898,-54.406,-177.595,5.899,148.332
C06877=1227.981,181.147,-54.429,-177.592,5.900,148.332
C06878=1227.975,181.396,-54.451,-177.589,5.902,148.331
C06879=1227.971,181.644,-54.474,-177.587,5.903,148.331
C06880=1227.967,181.893,-54.498,-177.585,5.905,148.330
C06881=1227.962,182.143,-54.520,-177.582,5.907,148.330
C06882=1227.957,182.391,-54.543,-177.579,5.907,148.329
C06883=1227.953,182.640,-54.565,-177.577,5.909,148.329
C06884=1227.948,182.889,-54.588,-177.575,5.910,148.329
C06885=1227.943,183.139,-54.611,-177.572,5.912,148.328
C06886=1227.939,183.387,-54.634,-177.569,5.913,148.328
C06887=1227.934,183.636,-54.657,-177.567,5.914,148.327
C06888=1227.929,183.885,-54.680,-177.564,5.916,148.327
C06889=1227.925,184.134,-54.702,-177.561,5.918,148.327
C06890=1227.921,184.383,-54.726,-177.559,5.919,148.326
C06891=1227.916,184.631,-54.748,-177.556,5.921,148.326
C06892=1227.911,184.880,-54.772,-177.554,5.922,148.325
C06893=1227.907,185.129,-54.795,-177.551,5.923,148.325
C06894=1227.902,185.398,-54.819,-177.549,5.925,148.325
C06895=1227.897,185.668,-54.844,-177.546,5.927,148.324
C06896=1227.891,185.938,-54.869,-177.543,5.929,148.324
C06897=1227.887,186.207,-54.894,-177.540,5.930,148.323
C06898=1227.882,186.457,-54.917,-177.537,5.932,148.323
C06899=1227.877,186.706,-54.941,-177.535,5.933,148.322
C06900=1227.873,186.955,-54.964,-177.532,5.935,148.322
C06901=1227.868,187.204,-54.986,-177.530,5.937,148.322
C06902=1227.863,187.452,-55.009,-177.527,5.937,148.321
C06903=1227.858,187.701,-55.032,-177.525,5.939,148.321
C06904=1227.854,187.950,-55.055,-177.522,5.941,148.320
C06905=1227.850,188.199,-55.079,-177.520,5.942,148.320
C06906=1227.845,188.448,-55.102,-177.517,5.944,148.320
C06907=1227.840,188.697,-55.125,-177.514,5.945,148.319
C06908=1227.836,188.946,-55.148,-177.512,5.946,148.319
C06909=1227.831,189.194,-55.171,-177.509,5.948,148.318
C06910=1227.826,189.443,-55.194,-177.507,5.950,148.318
C06911=1227.822,189.692,-55.218,-177.505,5.951,148.318
C06912=1227.817,189.941,-55.241,-177.502,5.953,148.317
C06913=1227.813,190.190,-55.264,-177.499,5.955,148.317
C06914=1227.808,190.439,-55.287,-177.497,5.956,148.316
C06915=1227.804,190.688,-55.311,-177.494,5.957,148.316
C06916=1227.799,190.937,-55.334,-177.492,5.959,148.316
C06917=1227.794,191.186,-55.357,-177.489,5.961,148.315
C06918=1227.790,191.435,-55.381,-177.486,5.962,148.315
C06919=1227.785,191.683,-55.404,-177.484,5.964,148.314
C06920=1227.781,191.932,-55.427,-177.481,5.965,148.314
C06921=1227.776,192.181,-55.450,-177.479,5.967,148.314
C06922=1227.771,192.430,-55.474,-177.476,5.968,148.313
C06923=1227.766,192.679,-55.497,-177.473,5.970,148.313
C06924=1227.762,192.928,-55.521,-177.471,5.972,148.312
C06925=1227.757,193.177,-55.544,-177.468,5.973,148.312
C06926=1227.753,193.425,-55.568,-177.466,5.975,148.312
C06927=1227.748,193.674,-55.591,-177.463,5.976,148.311
C06928=1227.744,193.923,-55.614,-177.461,5.977,148.311
C06929=1227.739,194.172,-55.637,-177.458,5.979,148.311
C06930=1227.735,194.421,-55.661,-177.455,5.981,148.310
C06931=1227.730,194.669,-55.685,-177.453,5.983,148.310
C06932=1227.725,194.918,-55.708,-177.451,5.984,148.309
C06933=1227.721,195.167,-55.732,-177.448,5.986,148.309
C06934=1227.716,195.416,-55.755,-177.445,5.987,148.309
C06935=1227.712,195.665,-55.779,-177.443,5.988,148.308
C06936=1227.707,195.914,-55.802,-177.440,5.990,148.308
C06937=1227.702,196.163,-55.826,-177.437,5.992,148.307
C06938=1227.698,196.412,-55.849,-177.435,5.994,148.307
C06939=1227.693,196.660,-55.873,-177.433,5.995,148.307
C06940=1227.689,196.909,-55.897,-177.430,5.996,148.306
C06941=1227.684,197.158,-55.920,-177.427,5.998,148.306
C06942=1227.679,197.407,-55.944,-177.425,6.000,148.306
C06943=1227.675,197.656,-55.967,-177.422,6.001,148.305
C06944=1227.670,197.905,-55.991,-177.420,6.003,148.305
C06945=1227.666,198.153,-56.015,-177.417,6.005,148.304
C06946=1227.661,198.402,-56.038,-177.414,6.006,148.304
C06947=1227.657,198.651,-56.062,-177.412,6.007,148.304
C06948=1227.652,198.900,-56.086,-177.410,6.009,148.303
C06949=1227.647,199.149,-56.109,-177.407,6.011,148.303
C06950=1227.643,199.397,-56.133,-177.404,6.013,148.302
C06951=1227.638,199.646,-56.156,-177.402,6.014,148.302
C06952=1227.634,199.895,-56.180,-177.399,6.016,148.302
C06953=1227.629,200.144,-56.204,-177.396,6.017,148.301
C06954=1227.624,200.392,-56.228,-177.394,6.019,148.301
C06955=1227.619,200.641,-56.252,-177.392,6.020,148.300
C06956=1227.615,200.891,-56.276,-177.389,6.022,148.300
C06957=1227.611,201.140,-56.300,-177.386,6.024,148.300
C06958=1227.606,201.388,-56.324,-177.384,6.026,148.299
C06959=1227.602,201.637,-56.347,-177.381,6.026,148.299
C06960=1227.597,201.886,-56.371,-177.379,6.028,148.299
C06961=1227.592,202.135,-56.394,-177.376,6.030,148.298
C06962=1227.588,202.383,-56.419,-177.373,6.032,148.298
C06963=1227.583,202.632,-56.442,-177.371,6.033,148.297
C06964=1227.578,202.881,-56.467,-177.369,6.035,148.297
C06965=1227.574,203.130,-56.490,-177.366,6.037,148.297
C06966=1227.570,203.379,-56.514,-177.363,6.039,148.296
C06967=1227.565,203.627,-56.538,-177.361,6.040,148.296
C06968=1227.561,203.876,-56.562,-177.359,6.042,148.296
C06969=1227.555,204.125,-56.586,-177.356,6.043,148.295
C06970=1227.551,204.374,-56.610,-177.353,6.045,148.295
C06971=1227.546,204.622,-56.634,-177.350,6.047,148.295
C06972=1227.542,204.871,-56.658,-177.348,6.049,148.294
C06973=1227.537,205.121,-56.682,-177.346,6.050,148.294
C06974=1227.533,205.369,-56.706,-177.343,6.051,148.293
C06975=1227.528,205.618,-56.730,-177.340,6.053,148.293
C06976=1227.524,205.867,-56.754,-177.338,6.055,148.293
C06977=1227.519,206.115,-56.778,-177.336,6.056,148.292
C06978=1227.514,206.364,-56.803,-177.333,6.058,148.292
C06979=1227.510,206.614,-56.826,-177.330,6.060,148.292
C06980=1227.506,206.862,-56.850,-177.327,6.061,148.291
C06981=1227.501,207.111,-56.875,-177.325,6.063,148.291
C06982=1227.496,207.359,-56.899,-177.322,6.065,148.291
C06983=1227.491,207.608,-56.922,-177.320,6.066,148.290
C06984=1227.488,207.857,-56.947,-177.317,6.068,148.290
C06985=1227.483,208.106,-56.972,-177.315,6.070,148.289
C06986=1227.478,208.354,-56.996,-177.312,6.072,148.289
C06987=1227.474,208.603,-57.020,-177.309,6.074,148.289
C06988=1227.468,208.852,-57.044,-177.307,6.075,148.288
C06989=1227.464,209.101,-57.068,-177.305,6.076,148.288
C06990=1227.460,209.350,-57.092,-177.302,6.078,148.288
C06991=1227.455,209.598,-57.117,-177.299,6.080,148.287
C06992=1227.451,209.847,-57.141,-177.297,6.082,148.287
C06993=1227.446,210.096,-57.166,-177.295,6.083,148.287
C06994=1227.442,210.345,-57.190,-177.292,6.085,148.286
C06995=1227.437,210.594,-57.213,-177.289,6.086,148.286
C06996=1227.432,210.842,-57.238,-177.286,6.088,148.286
C06997=1227.428,211.092,-57.263,-177.284,6.090,148.285
C06998=1227.423,211.362,-57.289,-177.281,6.092,148.285
C06999=1227.418,211.632,-57.316,-177.278,6.094,148.285
C07000=1227.413,211.902,-57.342,-177.276,6.096,148.284
C07001=1227.408,212.173,-57.368,-177.273,6.097,148.284
C07002=1227.403,212.422,-57.393,-177.270,6.099,148.283
C07003=1227.399,212.670,-57.417,-177.267,6.101,148.283
C07004=1227.394,212.919,-57.442,-177.265,6.103,148.283
C07005=1227.390,213.168,-57.466,-177.263,6.104,148.282
C07006=1227.385,213.417,-57.491,-177.260,6.106,148.282
C07007=1227.380,213.665,-57.515,-177.257,6.108,148.282
C07008=1227.377,213.915,-57.539,-177.255,6.109,148.281
C07009=1227.372,214.163,-57.564,-177.252,6.111,148.281
C07010=1227.367,214.412,-57.588,-177.249,6.113,148.281
C07011=1227.363,214.661,-57.613,-177.247,6.115,148.280
C07012=1227.359,214.909,-57.638,-177.245,6.116,148.280
C07013=1227.353,215.158,-57.663,-177.242,6.118,148.280
C07014=1227.350,215.407,-57.687,-177.240,6.120,148.279
C07015=1227.344,215.655,-57.712,-177.237,6.122,148.279
C07016=1227.339,215.904,-57.736,-177.234,6.124,148.279
C07017=1227.336,216.153,-57.761,-177.232,6.125,148.278
C07018=1227.330,216.402,-57.786,-177.229,6.127,148.278
C07019=1227.326,216.650,-57.810,-177.227,6.128,148.278
C07020=1227.322,216.899,-57.835,-177.224,6.130,148.277
C07021=1227.317,217.148,-57.859,-177.222,6.132,148.277
C07022=1227.312,217.396,-57.884,-177.219,6.134,148.277
C07023=1227.308,217.645,-57.909,-177.216,6.136,148.276
C07024=1227.303,217.894,-57.933,-177.214,6.138,148.276
C07025=1227.299,218.143,-57.959,-177.211,6.139,148.276
C07026=1227.295,218.391,-57.983,-177.209,6.141,148.275
C07027=1227.290,218.640,-58.008,-177.206,6.142,148.275
C07028=1227.286,218.889,-58.032,-177.204,6.144,148.275
C07029=1227.281,219.137,-58.058,-177.201,6.146,148.274
C07030=1227.276,219.387,-58.083,-177.199,6.148,148.274
C07031=1227.272,219.635,-58.107,-177.196,6.150,148.274
C07032=1227.267,219.884,-58.131,-177.193,6.152,148.273
C07033=1227.263,220.133,-58.157,-177.191,6.154,148.273
C07034=1227.258,220.381,-58.181,-177.188,6.155,148.273
C07035=1227.254,220.631,-58.206,-177.186,6.156,148.272
C07036=1227.249,220.879,-58.232,-177.183,6.158,148.272
C07037=1227.245,221.128,-58.256,-177.181,6.160,148.272
C07038=1227.240,221.376,-58.281,-177.178,6.162,148.271
C07039=1227.235,221.625,-58.306,-177.175,6.164,148.271
C07040=1227.231,221.874,-58.331,-177.173,6.166,148.271
C07041=1227.226,222.122,-58.355,-177.170,6.168,148.270
C07042=1227.222,222.371,-58.381,-177.168,6.169,148.270
C07043=1227.217,222.620,-58.406,-177.165,6.171,148.270
C07044=1227.213,222.868,-58.431,-177.163,6.172,148.269
C07045=1227.208,223.117,-58.455,-177.160,6.174,148.269
C07046=1227.204,223.366,-58.481,-177.158,6.176,148.269
C07047=1227.200,223.614,-58.505,-177.155,6.178,148.268
C07048=1227.195,223.863,-58.531,-177.152,6.180,148.268
C07049=1227.190,224.112,-58.556,-177.150,6.182,148.268
C07050=1227.186,224.361,-58.581,-177.147,6.184,148.267
C07051=1227.181,224.609,-58.606,-177.145,6.185,148.267
C07052=1227.177,224.859,-58.631,-177.142,6.187,148.267
C07053=1227.172,225.107,-58.656,-177.139,6.189,148.266
C07054=1227.168,225.355,-58.682,-177.137,6.190,148.266
C07055=1227.163,225.604,-58.706,-177.135,6.192,148.266
C07056=1227.159,225.853,-58.732,-177.132,6.194,148.266
C07057=1227.154,226.101,-58.756,-177.130,6.196,148.265
C07058=1227.150,226.350,-58.782,-177.127,6.198,148.265
C07059=1227.145,226.599,-58.807,-177.125,6.200,148.265
C07060=1227.141,226.848,-58.832,-177.122,6.202,148.264
C07061=1227.136,227.096,-58.858,-177.119,6.204,148.264
C07062=1227.131,227.345,-58.883,-177.117,6.205,148.264
C07063=1227.127,227.593,-58.908,-177.114,6.207,148.263
C07064=1227.123,227.842,-58.933,-177.112,6.208,148.263
C07065=1227.119,228.091,-58.958,-177.109,6.210,148.263
C07066=1227.114,228.339,-58.984,-177.107,6.212,148.262
C07067=1227.109,228.589,-59.009,-177.104,6.214,148.262
C07068=1227.104,228.837,-59.034,-177.102,6.216,148.262
C07069=1227.100,229.086,-59.060,-177.099,6.218,148.262
C07070=1227.095,229.334,-59.085,-177.097,6.220,148.261
C07071=1227.091,229.583,-59.110,-177.094,6.222,148.261
C07072=1227.087,229.832,-59.136,-177.092,6.224,148.261
C07073=1227.082,230.080,-59.161,-177.089,6.226,148.260
C07074=1227.077,230.330,-59.186,-177.086,6.227,148.260
C07075=1227.072,230.578,-59.212,-177.084,6.229,148.260
C07076=1227.069,230.826,-59.237,-177.081,6.231,148.259
C07077=1227.065,231.075,-59.263,-177.079,6.232,148.259
C07078=1227.060,231.324,-59.287,-177.076,6.234,148.259
C07079=1227.055,231.573,-59.313,-177.074,6.236,148.258
C07080=1227.051,231.821,-59.339,-177.072,6.238,148.258
C07081=1227.046,232.069,-59.364,-177.069,6.240,148.258
C07082=1227.042,232.318,-59.390,-177.066,6.242,148.258
C07083=1227.037,232.566,-59.415,-177.064,6.244,148.257
C07084=1227.033,232.816,-59.441,-177.061,6.246,148.257
C07085=1227.028,233.065,-59.466,-177.058,6.247,148.257
C07086=1227.024,233.313,-59.492,-177.056,6.249,148.256
C07087=1227.019,233.562,-59.518,-177.053,6.251,148.256
C07088=1227.014,233.811,-59.544,-177.051,6.253,148.256
C07089=1227.010,234.059,-59.569,-177.048,6.255,148.256
C07090=1227.005,234.307,-59.595,-177.046,6.257,148.255
C07091=1227.001,234.556,-59.621,-177.043,6.259,148.255
C07092=1226.996,234.804,-59.646,-177.041,6.260,148.255
C07093=1226.992,235.053,-59.672,-177.039,6.262,148.254
C07094=1226.988,235.303,-59.697,-177.036,6.264,148.254
C07095=1226.983,235.551,-59.722,-177.033,6.266,148.254
C07096=1226.979,235.800,-59.748,-177.031,6.268,148.253
C07097=1226.974,236.048,-59.774,-177.029,6.270,148.253
C07098=1226.970,236.297,-59.799,-177.026,6.272,148.253
C07099=1226.965,236.546,-59.825,-177.023,6.273,148.253
C07100=1226.960,236.794,-59.851,-177.021,6.275,148.252
C07101=1226.956,237.043,-59.878,-177.018,6.277,148.252
C07102=1226.951,237.314,-59.905,-177.015,6.279,148.252
C07103=1226.946,237.586,-59.933,-177.012,6.282,148.251
C07104=1226.941,237.857,-59.961,-177.010,6.284,148.251
C07105=1226.937,238.128,-59.990,-177.007,6.286,148.251
C07106=1226.933,238.377,-60.016,-177.004,6.287,148.250
C07107=1226.928,238.626,-60.041,-177.002,6.289,148.250
C07108=1226.923,238.874,-60.067,-177.000,6.292,148.250
C07109=1226.919,239.123,-60.093,-176.997,6.293,148.250
C07110=1226.914,239.372,-60.119,-176.994,6.295,148.249
C07111=1226.910,239.620,-60.145,-176.992,6.297,148.249
C07112=1226.905,239.868,-60.171,-176.989,6.299,148.249
C07113=1226.901,240.117,-60.197,-176.987,6.301,148.248
C07114=1226.896,240.366,-60.223,-176.984,6.303,148.248
C07115=1226.892,240.615,-60.248,-176.982,6.305,148.248
C07116=1226.887,240.863,-60.275,-176.979,6.307,148.248
C07117=1226.883,241.111,-60.301,-176.977,6.309,148.247
C07118=1226.878,241.360,-60.327,-176.974,6.311,148.247
C07119=1226.874,241.609,-60.352,-176.972,6.313,148.247
C07120=1226.869,241.858,-60.379,-176.969,6.315,148.247
C07121=1226.865,242.106,-60.405,-176.967,6.317,148.246
C07122=1226.860,242.354,-60.431,-176.964,6.318,148.246
C07123=1226.856,242.603,-60.456,-176.961,6.320,148.246
C07124=1226.852,242.852,-60.483,-176.959,6.322,148.245
C07125=1226.847,243.100,-60.509,-176.957,6.324,148.245
C07126=1226.843,243.349,-60.535,-176.955,6.325,148.245
C07127=1226.838,243.598,-60.561,-176.952,6.327,148.245
C07128=1226.834,243.846,-60.587,-176.949,6.329,148.244
C07129=1226.829,244.095,-60.613,-176.947,6.331,148.244
C07130=1226.825,244.343,-60.640,-176.945,6.333,148.244
C07131=1226.821,244.592,-60.666,-176.942,6.335,148.244
C07132=1226.816,244.841,-60.692,-176.939,6.337,148.243
C07133=1226.812,245.089,-60.719,-176.937,6.339,148.243
C07134=1226.807,245.337,-60.744,-176.935,6.341,148.243
C07135=1226.802,245.587,-60.770,-176.932,6.343,148.243
C07136=1226.798,245.835,-60.797,-176.929,6.345,148.242
C07137=1226.793,246.084,-60.823,-176.927,6.347,148.242
C07138=1226.789,246.332,-60.850,-176.924,6.349,148.242
C07139=1226.785,246.581,-60.876,-176.922,6.352,148.242
C07140=1226.780,246.829,-60.903,-176.919,6.353,148.241
C07141=1226.776,247.078,-60.928,-176.916,6.355,148.241
C07142=1226.771,247.327,-60.955,-176.914,6.357,148.241
C07143=1226.767,247.575,-60.981,-176.912,6.359,148.241
C07144=1226.762,247.823,-61.008,-176.909,6.361,148.240
C07145=1226.758,248.072,-61.034,-176.906,6.363,148.240
C07146=1226.754,248.320,-61.060,-176.904,6.365,148.240
C07147=1226.749,248.569,-61.086,-176.902,6.367,148.240
C07148=1226.745,248.817,-61.113,-176.899,6.369,148.239
C07149=1226.740,249.067,-61.139,-176.896,6.371,148.239
C07150=1226.736,249.315,-61.166,-176.894,6.373,148.239
C07151=1226.731,249.563,-61.193,-176.892,6.375,148.239
C07152=1226.727,249.812,-61.218,-176.889,6.377,148.238
C07153=1226.722,250.061,-61.246,-176.886,6.379,148.238
C07154=1226.717,250.310,-61.272,-176.884,6.381,148.238
C07155=1226.714,250.558,-61.298,-176.882,6.383,148.237
C07156=1226.709,250.806,-61.325,-176.879,6.385,148.237
C07157=1226.705,251.055,-61.351,-176.876,6.387,148.237
C07158=1226.700,251.304,-61.378,-176.874,6.389,148.237
C07159=1226.696,251.552,-61.405,-176.872,6.391,148.236
C07160=1226.691,251.801,-61.431,-176.869,6.393,148.236
C07161=1226.687,252.048,-61.457,-176.867,6.395,148.236
C07162=1226.682,252.297,-61.484,-176.864,6.396,148.236
C07163=1226.677,252.546,-61.511,-176.862,6.399,148.235
C07164=1226.673,252.794,-61.537,-176.859,6.401,148.235
C07165=1226.668,253.043,-61.564,-176.857,6.402,148.235
C07166=1226.665,253.292,-61.591,-176.854,6.405,148.235
C07167=1226.660,253.541,-61.617,-176.852,6.407,148.234
C07168=1226.655,253.789,-61.644,-176.849,6.408,148.234
C07169=1226.652,254.037,-61.671,-176.847,6.410,148.234
C07170=1226.647,254.286,-61.698,-176.844,6.413,148.234
C07171=1226.642,254.534,-61.725,-176.841,6.415,148.234
C07172=1226.638,254.783,-61.751,-176.839,6.417,148.233
C07173=1226.633,255.032,-61.778,-176.837,6.419,148.233
C07174=1226.629,255.280,-61.805,-176.834,6.421,148.233
C07175=1226.625,255.528,-61.831,-176.831,6.423,148.233
C07176=1226.620,255.777,-61.858,-176.829,6.425,148.232
C07177=1226.615,256.025,-61.885,-176.827,6.427,148.232
C07178=1226.612,256.274,-61.912,-176.824,6.429,148.232
C07179=1226.607,256.522,-61.939,-176.821,6.431,148.232
C07180=1226.602,256.771,-61.965,-176.819,6.433,148.231
C07181=1226.597,257.020,-61.992,-176.817,6.435,148.231
C07182=1226.593,257.268,-62.019,-176.814,6.437,148.231
C07183=1226.589,257.516,-62.046,-176.812,6.439,148.231
C07184=1226.584,257.765,-62.073,-176.809,6.441,148.230
C07185=1226.580,258.014,-62.100,-176.806,6.444,148.230
C07186=1226.576,258.262,-62.127,-176.804,6.446,148.230
C07187=1226.571,258.511,-62.154,-176.801,6.448,148.230
C07188=1226.567,258.759,-62.181,-176.799,6.450,148.229
C07189=1226.562,259.008,-62.208,-176.797,6.452,148.229
C07190=1226.558,259.256,-62.234,-176.794,6.454,148.229
C07191=1226.554,259.504,-62.261,-176.791,6.456,148.229
C07192=1226.549,259.753,-62.289,-176.789,6.458,148.229
C07193=1226.544,260.001,-62.316,-176.787,6.460,148.228
C07194=1226.540,260.251,-62.343,-176.784,6.462,148.228
C07195=1226.535,260.499,-62.370,-176.782,6.464,148.228
C07196=1226.532,260.747,-62.397,-176.779,6.467,148.228
C07197=1226.527,260.995,-62.424,-176.776,6.468,148.227
C07198=1226.523,261.244,-62.451,-176.774,6.471,148.227
C07199=1226.518,261.492,-62.478,-176.772,6.473,148.227
C07200=1226.514,261.741,-62.506,-176.769,6.475,148.227
C07201=1226.509,261.990,-62.533,-176.767,6.477,148.227
C07202=1226.505,262.238,-62.560,-176.764,6.478,148.226
C07203=1226.501,262.487,-62.586,-176.762,6.481,148.226
C07204=1226.496,262.734,-62.614,-176.759,6.483,148.226
C07205=1226.492,262.983,-62.641,-176.757,6.484,148.226
C07206=1226.486,263.256,-62.672,-176.754,6.488,148.226
C07207=1226.482,263.529,-62.701,-176.752,6.489,148.225
C07208=1226.477,263.802,-62.731,-176.748,6.492,148.225
C07209=1226.472,264.074,-62.761,-176.746,6.494,148.225
C07210=1226.468,264.323,-62.788,-176.744,6.496,148.225
C07211=1226.463,264.570,-62.816,-176.741,6.498,148.224
C07212=1226.459,264.819,-62.843,-176.739,6.500,148.224
C07213=1226.455,265.068,-62.870,-176.736,6.503,148.224
C07214=1226.450,265.317,-62.897,-176.733,6.505,148.224
C07215=1226.446,265.565,-62.925,-176.731,6.507,148.224
C07216=1226.441,265.813,-62.952,-176.728,6.509,148.223
C07217=1226.437,266.062,-62.980,-176.726,6.511,148.223
C07218=1226.433,266.310,-63.007,-176.724,6.513,148.223
C07219=1226.428,266.559,-63.035,-176.721,6.515,148.223
C07220=1226.423,266.807,-63.062,-176.719,6.517,148.223
C07221=1226.419,267.056,-63.090,-176.716,6.520,148.222
C07222=1226.415,267.304,-63.117,-176.714,6.522,148.222
C07223=1226.410,267.552,-63.145,-176.711,6.524,148.222
C07224=1226.406,267.801,-63.172,-176.709,6.526,148.222
C07225=1226.402,268.050,-63.199,-176.706,6.528,148.222
C07226=1226.397,268.298,-63.227,-176.704,6.530,148.221
C07227=1226.393,268.546,-63.254,-176.702,6.532,148.221
C07228=1226.388,268.794,-63.282,-176.699,6.535,148.221
C07229=1226.384,269.043,-63.309,-176.696,6.537,148.221
C07230=1226.380,269.291,-63.337,-176.694,6.539,148.221
C07231=1226.375,269.540,-63.364,-176.691,6.541,148.220
C07232=1226.371,269.788,-63.393,-176.689,6.543,148.220
C07233=1226.366,270.037,-63.420,-176.687,6.545,148.220
C07234=1226.362,270.285,-63.448,-176.684,6.547,148.220
C07235=1226.358,270.534,-63.475,-176.681,6.550,148.220
C07236=1226.353,270.782,-63.503,-176.679,6.552,148.220
C07237=1226.349,271.030,-63.530,-176.677,6.554,148.219
C07238=1226.345,271.279,-63.558,-176.674,6.556,148.219
C07239=1226.340,271.528,-63.586,-176.672,6.558,148.219
C07240=1226.335,271.776,-63.613,-176.670,6.560,148.219
C07241=1226.332,272.024,-63.642,-176.667,6.563,148.219
C07242=1226.327,272.273,-63.669,-176.664,6.565,148.218
C07243=1226.323,272.521,-63.696,-176.662,6.567,148.218
C07244=1226.319,272.769,-63.724,-176.659,6.569,148.218
C07245=1226.313,273.018,-63.752,-176.657,6.571,148.218
C07246=1226.309,273.266,-63.780,-176.655,6.573,148.218
C07247=1226.305,273.515,-63.807,-176.652,6.576,148.218
C07248=1226.301,273.763,-63.835,-176.649,6.578,148.217
C07249=1226.296,274.012,-63.864,-176.647,6.580,148.217
C07250=1226.292,274.260,-63.892,-176.645,6.582,148.217
C07251=1226.287,274.508,-63.919,-176.642,6.584,148.217
C07252=1226.283,274.757,-63.947,-176.640,6.586,148.217
C07253=1226.278,275.005,-63.975,-176.637,6.589,148.217
C07254=1226.274,275.254,-64.003,-176.635,6.591,148.216
C07255=1226.270,275.502,-64.030,-176.632,6.593,148.216
C07256=1226.266,275.750,-64.058,-176.630,6.595,148.216
C07257=1226.261,275.999,-64.087,-176.628,6.598,148.216
C07258=1226.257,276.247,-64.115,-176.625,6.600,148.216
C07259=1226.253,276.496,-64.142,-176.622,6.603,148.216
C07260=1226.248,276.744,-64.171,-176.620,6.604,148.215
C07261=1226.244,276.993,-64.199,-176.618,6.607,148.215
C07262=1226.239,277.240,-64.226,-176.616,6.609,148.215
C07263=1226.234,277.489,-64.255,-176.612,6.612,148.215
C07264=1226.231,277.737,-64.283,-176.610,6.614,148.215
C07265=1226.226,277.986,-64.310,-176.608,6.616,148.214
C07266=1226.221,278.235,-64.339,-176.606,6.618,148.214
C07267=1226.217,278.482,-64.367,-176.603,6.620,148.214
C07268=1226.213,278.731,-64.395,-176.600,6.623,148.214
C07269=1226.208,278.979,-64.423,-176.598,6.625,148.214
C07270=1226.205,279.228,-64.451,-176.596,6.627,148.214
C07271=1226.200,279.476,-64.479,-176.593,6.629,148.213
C07272=1226.196,279.725,-64.508,-176.591,6.631,148.213
C07273=1226.191,279.972,-64.535,-176.588,6.634,148.213
C07274=1226.187,280.221,-64.564,-176.586,6.636,148.213
C07275=1226.182,280.469,-64.592,-176.584,6.638,148.213
C07276=1226.178,280.718,-64.621,-176.581,6.640,148.213
C07277=1226.174,280.966,-64.648,-176.579,6.642,148.213
C07278=1226.170,281.215,-64.677,-176.576,6.645,148.212
C07279=1226.165,281.463,-64.705,-176.574,6.647,148.212
C07280=1226.161,281.711,-64.733,-176.571,6.649,148.212
C07281=1226.156,281.960,-64.762,-176.569,6.651,148.212
C07282=1226.152,282.208,-64.790,-176.566,6.654,148.212
C07283=1226.147,282.456,-64.818,-176.564,6.656,148.212
C07284=1226.143,282.705,-64.846,-176.561,6.659,148.212
C07285=1226.138,282.953,-64.875,-176.559,6.661,148.212
C07286=1226.135,283.202,-64.903,-176.557,6.663,148.211
C07287=1226.130,283.449,-64.932,-176.554,6.666,148.211
C07288=1226.126,283.698,-64.960,-176.552,6.668,148.211
C07289=1226.122,283.947,-64.989,-176.549,6.670,148.211
C07290=1226.117,284.195,-65.016,-176.547,6.672,148.211
C07291=1226.113,284.443,-65.045,-176.544,6.675,148.211
C07292=1226.108,284.691,-65.073,-176.542,6.677,148.211
C07293=1226.104,284.940,-65.102,-176.540,6.679,148.210
C07294=1226.099,285.188,-65.131,-176.537,6.681,148.210
C07295=1226.095,285.436,-65.159,-176.535,6.684,148.210
C07296=1226.091,285.685,-65.188,-176.532,6.686,148.210
C07297=1226.086,285.933,-65.215,-176.530,6.688,148.210
C07298=1226.082,286.181,-65.245,-176.528,6.690,148.210
C07299=1226.077,286.430,-65.273,-176.525,6.692,148.209
C07300=1226.073,286.678,-65.301,-176.523,6.695,148.209
C07301=1226.069,286.927,-65.330,-176.520,6.698,148.209
C07302=1226.065,287.174,-65.359,-176.518,6.699,148.209
C07303=1226.060,287.423,-65.387,-176.516,6.702,148.209
C07304=1226.056,287.672,-65.416,-176.513,6.705,148.209
C07305=1226.052,287.919,-65.445,-176.510,6.707,148.209
C07306=1226.047,288.168,-65.473,-176.508,6.709,148.209
C07307=1226.042,288.416,-65.502,-176.506,6.711,148.209
C07308=1226.039,288.664,-65.531,-176.503,6.714,148.208
C07309=1226.034,288.913,-65.559,-176.501,6.716,148.208
